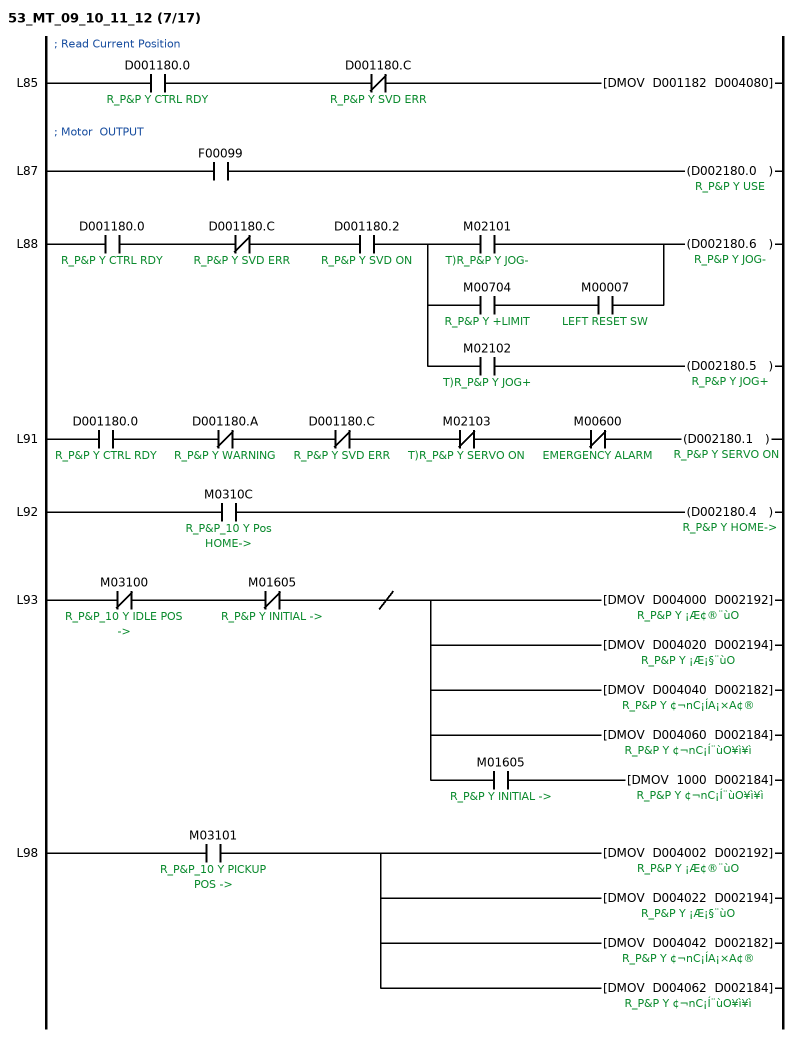
[picture p288: 53_MT_09_10_11_12 rungs L85-L98]
; L85
LOAD      D001180.0	// R_P&P Y CTRL RDY
AND NOT   D001180.C	// R_P&P Y SVD ERR
DMOV      D001182 D004080
// output comment: Read Current Position
//  Motor  OUTPUT
; L87
LOAD      F00099
OUT       D002180.0	// R_P&P Y USE
; L88
LOAD      D001180.0	// R_P&P Y CTRL RDY
AND NOT   D001180.C	// R_P&P Y SVD ERR
AND       D001180.2	// R_P&P Y SVD ON
MPUSH
LOAD      M02101	// T)R_P&P Y JOG-
LOAD      M00704	// R_P&P Y +LIMIT
AND       M00007	// LEFT RESET SW
OR LOAD
AND LOAD
OUT       D002180.6	// R_P&P Y JOG-
MPOP
AND       M02102	// T)R_P&P Y JOG+
OUT       D002180.5	// R_P&P Y JOG+
; L91
LOAD      D001180.0	// R_P&P Y CTRL RDY
AND NOT   D001180.A	// R_P&P Y WARNING
AND NOT   D001180.C	// R_P&P Y SVD ERR
AND NOT   M02103	// T)R_P&P Y SERVO ON
AND NOT   M00600	// EMERGENCY ALARM
OUT       D002180.1	// R_P&P Y SERVO ON
; L92
LOAD      M0310C	// R_P&P_10 Y Pos HOME->
OUT       D002180.4	// R_P&P Y HOME->
; L93
LOAD NOT  M03100	// R_P&P_10 Y IDLE POS ->
AND NOT   M01605	// R_P&P Y INITIAL ->
NOT
DMOV      D004000 D002192	// R_P&P Y ¡Æ¢®¨ùO
DMOV      D004020 D002194	// R_P&P Y ¡Æ¡§¨ùO
DMOV      D004040 D002182	// R_P&P Y ¢¬nC¡ÍA¡×A¢®
DMOV      D004060 D002184	// R_P&P Y ¢¬nC¡Í¨ùO¥ì¥ì
AND       M01605	// R_P&P Y INITIAL ->
DMOV      1000 D002184	// R_P&P Y ¢¬nC¡Í¨ùO¥ì¥ì
; L98
LOAD      M03101	// R_P&P_10 Y PICKUP POS ->
DMOV      D004002 D002192	// R_P&P Y ¡Æ¢®¨ùO
DMOV      D004022 D002194	// R_P&P Y ¡Æ¡§¨ùO
DMOV      D004042 D002182	// R_P&P Y ¢¬nC¡ÍA¡×A¢®
DMOV      D004062 D002184	// R_P&P Y ¢¬nC¡Í¨ùO¥ì¥ì

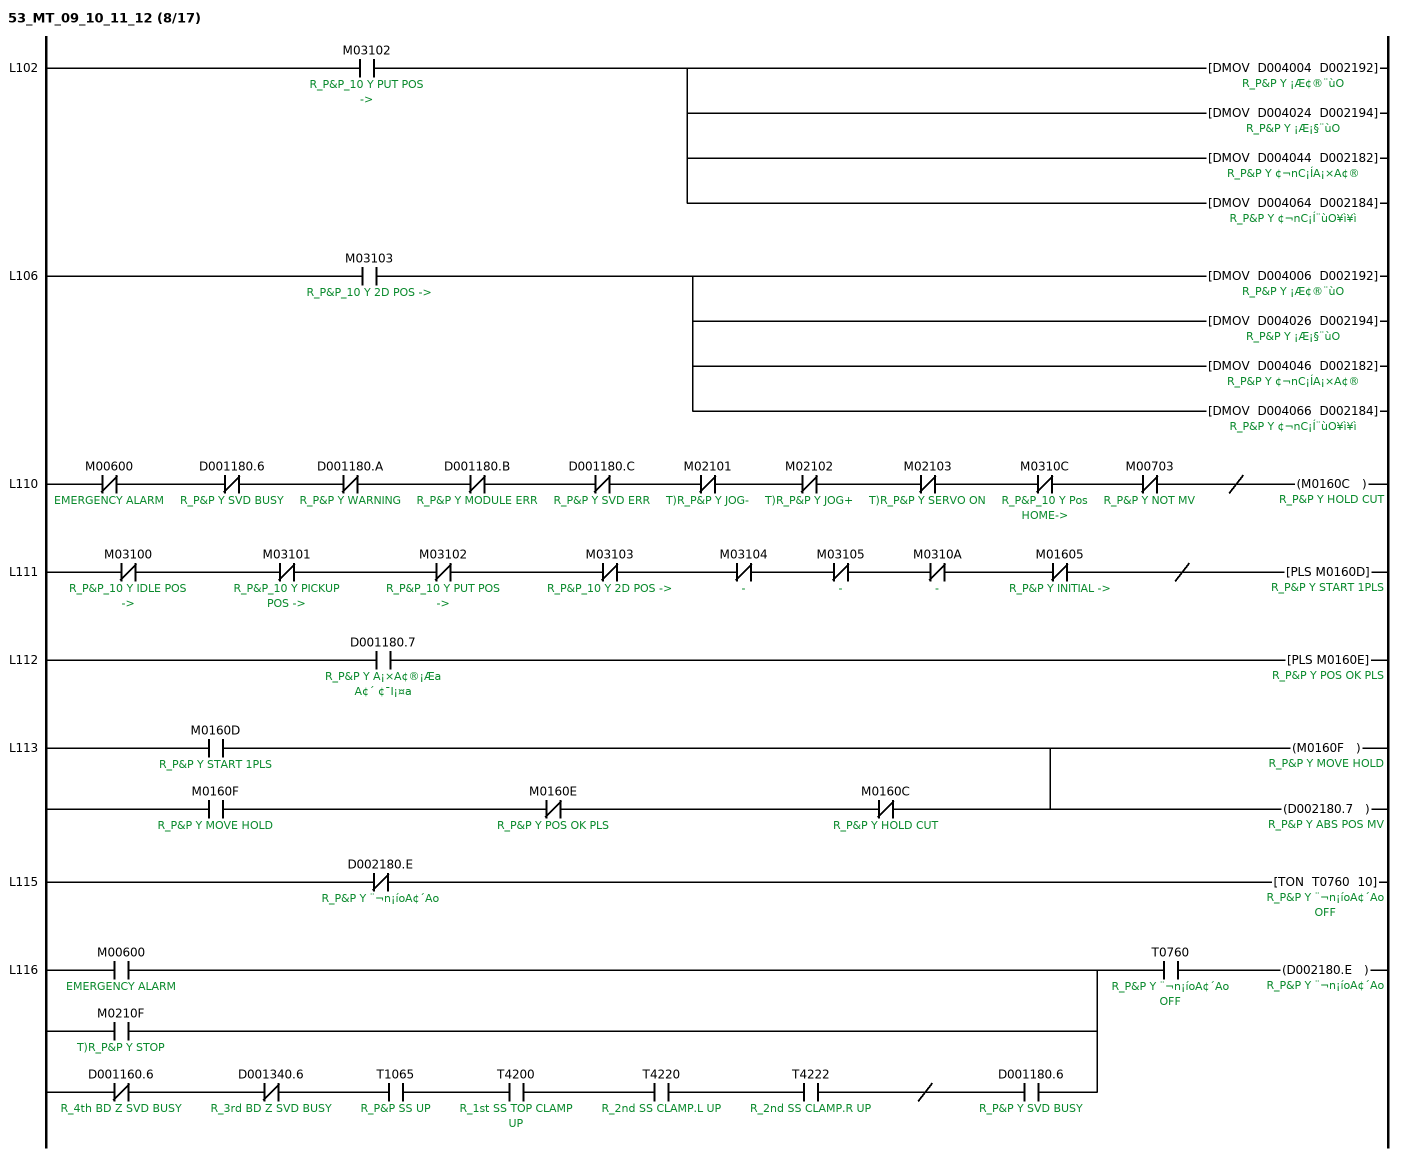
; L102
LOAD      M03102	// R_P&P_10 Y PUT POS ->
DMOV      D004004 D002192	// R_P&P Y ¡Æ¢®¨ùO
DMOV      D004024 D002194	// R_P&P Y ¡Æ¡§¨ùO
DMOV      D004044 D002182	// R_P&P Y ¢¬nC¡ÍA¡×A¢®
DMOV      D004064 D002184	// R_P&P Y ¢¬nC¡Í¨ùO¥ì¥ì
; L106
LOAD      M03103	// R_P&P_10 Y 2D POS ->
DMOV      D004006 D002192	// R_P&P Y ¡Æ¢®¨ùO
DMOV      D004026 D002194	// R_P&P Y ¡Æ¡§¨ùO
DMOV      D004046 D002182	// R_P&P Y ¢¬nC¡ÍA¡×A¢®
DMOV      D004066 D002184	// R_P&P Y ¢¬nC¡Í¨ùO¥ì¥ì
; L110
LOAD NOT  M00600	// EMERGENCY ALARM
AND NOT   D001180.6	// R_P&P Y SVD BUSY
AND NOT   D001180.A	// R_P&P Y WARNING
AND NOT   D001180.B	// R_P&P Y MODULE ERR
AND NOT   D001180.C	// R_P&P Y SVD ERR
AND NOT   M02101	// T)R_P&P Y JOG-
AND NOT   M02102	// T)R_P&P Y JOG+
AND NOT   M02103	// T)R_P&P Y SERVO ON
AND NOT   M0310C	// R_P&P_10 Y Pos HOME->
AND NOT   M00703	// R_P&P Y NOT MV
NOT
OUT       M0160C	// R_P&P Y HOLD CUT
; L111
LOAD NOT  M03100	// R_P&P_10 Y IDLE POS ->
AND NOT   M03101	// R_P&P_10 Y PICKUP POS ->
AND NOT   M03102	// R_P&P_10 Y PUT POS ->
AND NOT   M03103	// R_P&P_10 Y 2D POS ->
AND NOT   M03104	// -
AND NOT   M03105	// -
AND NOT   M0310A	// -
AND NOT   M01605	// R_P&P Y INITIAL ->
NOT
OUTP      M0160D	// R_P&P Y START 1PLS
; L112
LOAD      D001180.7	// R_P&P Y A¡×A¢®¡ÆaA¢´ ¢¯I¡¤a
OUTP      M0160E	// R_P&P Y POS OK PLS
; L113
LOAD      M0160D	// R_P&P Y START 1PLS
LOAD      M0160F	// R_P&P Y MOVE HOLD
AND NOT   M0160E	// R_P&P Y POS OK PLS
AND NOT   M0160C	// R_P&P Y HOLD CUT
OR LOAD
OUT       M0160F	// R_P&P Y MOVE HOLD
OUT       D002180.7	// R_P&P Y ABS POS MV
; L115
LOAD NOT  D002180.E	// R_P&P Y ¨¬n¡íoA¢´Ao
TON       T0760 10	// R_P&P Y ¨¬n¡íoA¢´AoOFF
; L116
LOAD      M00600	// EMERGENCY ALARM
OR        M0210F	// T)R_P&P Y STOP
LOAD NOT  D001160.6	// R_4th BD Z SVD BUSY
AND NOT   D001340.6	// R_3rd BD Z SVD BUSY
AND       T1065	// R_P&P SS UP
AND       T4200	// R_1st SS TOP CLAMP UP
AND       T4220	// R_2nd SS CLAMP.L UP
AND       T4222	// R_2nd SS CLAMP.R UP
NOT
AND       D001180.6	// R_P&P Y SVD BUSY
OR LOAD
AND       T0760	// R_P&P Y ¨¬n¡íoA¢´AoOFF
OUT       D002180.E	// R_P&P Y ¨¬n¡íoA¢´Ao

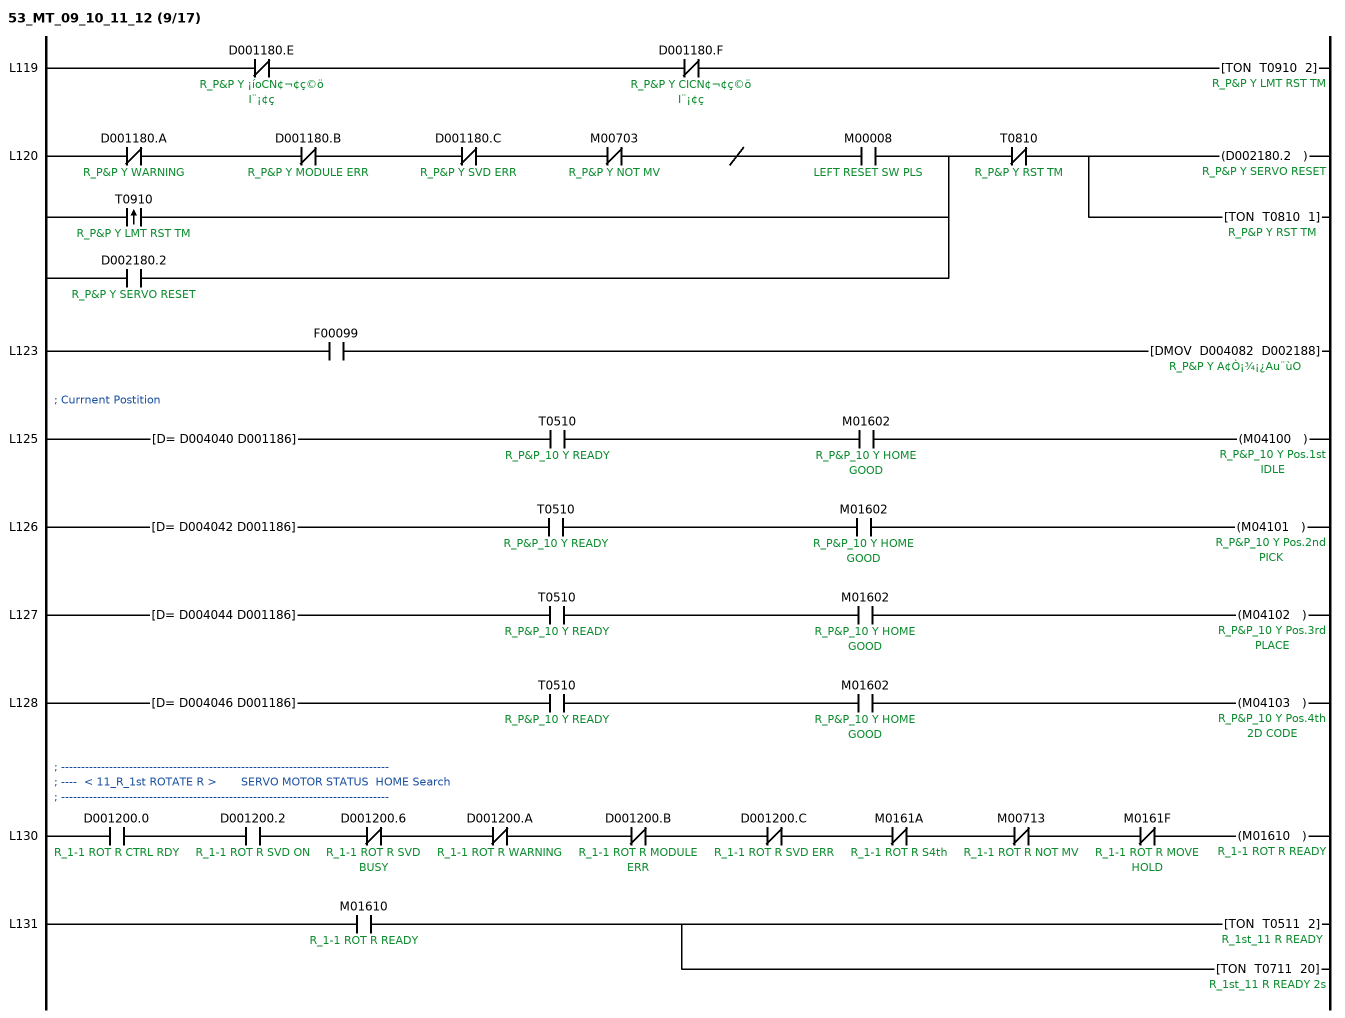
; L119
LOAD NOT  D001180.E	// R_P&P Y ¡íoCN¢¬¢ç©öI¨¡¢ç
AND NOT   D001180.F	// R_P&P Y CICN¢¬¢ç©öI¨¡¢ç
TON       T0910 2	// R_P&P Y LMT RST TM
; L120
LOAD NOT  D001180.A	// R_P&P Y WARNING
AND NOT   D001180.B	// R_P&P Y MODULE ERR
AND NOT   D001180.C	// R_P&P Y SVD ERR
AND NOT   M00703	// R_P&P Y NOT MV
NOT
AND       M00008	// LEFT RESET SW PLS
ORP       T0910	// R_P&P Y LMT RST TM
OR        D002180.2	// R_P&P Y SERVO RESET
AND NOT   T0810	// R_P&P Y RST TM
OUT       D002180.2	// R_P&P Y SERVO RESET
TON       T0810 1	// R_P&P Y RST TM
; L123
LOAD      F00099
DMOV      D004082 D002188	// R_P&P Y A¢Ò¡¾¡¿Au¨ùO
// Currnent Postition
; L125
LOADD=    D004040 D001186
AND       T0510	// R_P&P_10 Y READY
AND       M01602	// R_P&P_10 Y HOME GOOD
OUT       M04100	// R_P&P_10 Y Pos.1st IDLE
; L126
LOADD=    D004042 D001186
AND       T0510	// R_P&P_10 Y READY
AND       M01602	// R_P&P_10 Y HOME GOOD
OUT       M04101	// R_P&P_10 Y Pos.2nd PICK
; L127
LOADD=    D004044 D001186
AND       T0510	// R_P&P_10 Y READY
AND       M01602	// R_P&P_10 Y HOME GOOD
OUT       M04102	// R_P&P_10 Y Pos.3rd PLACE
; L128
LOADD=    D004046 D001186
AND       T0510	// R_P&P_10 Y READY
AND       M01602	// R_P&P_10 Y HOME GOOD
OUT       M04103	// R_P&P_10 Y Pos.4th 2D CODE
// ----------------------------------------------------------------------------------
// 
// ----  < 11_R_1st ROTATE R >       SERVO MOTOR STATUS  HOME Search
// 
// ----------------------------------------------------------------------------------
; L130
LOAD      D001200.0	// R_1-1 ROT R CTRL RDY
AND       D001200.2	// R_1-1 ROT R SVD ON
AND NOT   D001200.6	// R_1-1 ROT R SVD BUSY
AND NOT   D001200.A	// R_1-1 ROT R WARNING
AND NOT   D001200.B	// R_1-1 ROT R MODULE ERR
AND NOT   D001200.C	// R_1-1 ROT R SVD ERR
AND NOT   M0161A	// R_1-1 ROT R S4th
AND NOT   M00713	// R_1-1 ROT R NOT MV
AND NOT   M0161F	// R_1-1 ROT R MOVE HOLD
OUT       M01610	// R_1-1 ROT R READY
; L131
LOAD      M01610	// R_1-1 ROT R READY
TON       T0511 2	// R_1st_11 R READY
TON       T0711 20	// R_1st_11 R READY 2s

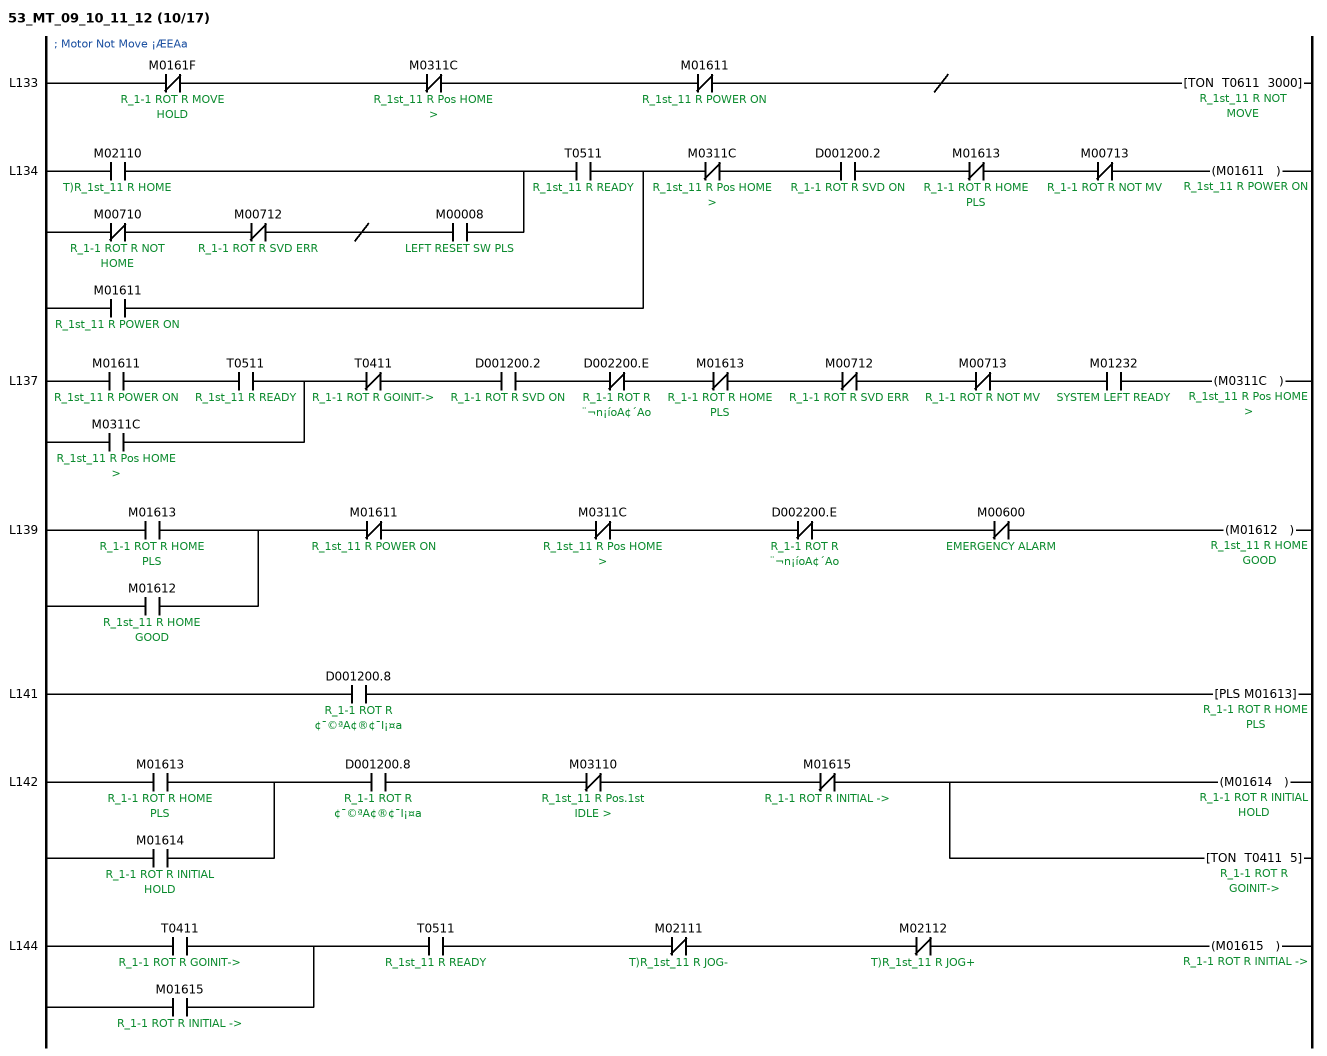
; L133
LOAD NOT  M0161F	// R_1-1 ROT R MOVE HOLD
AND NOT   M0311C	// R_1st_11 R Pos HOME >
AND NOT   M01611	// R_1st_11 R POWER ON
NOT
TON       T0611 3000	// R_1st_11 R NOT MOVE
// output comment: Motor Not Move ¡ÆEAa
; L134
LOAD      M02110	// T)R_1st_11 R HOME
LOAD NOT  M00710	// R_1-1 ROT R NOT HOME
AND NOT   M00712	// R_1-1 ROT R SVD ERR
NOT
AND       M00008	// LEFT RESET SW PLS
OR LOAD
AND       T0511	// R_1st_11 R READY
OR        M01611	// R_1st_11 R POWER ON
AND NOT   M0311C	// R_1st_11 R Pos HOME >
AND       D001200.2	// R_1-1 ROT R SVD ON
AND NOT   M01613	// R_1-1 ROT R HOME PLS
AND NOT   M00713	// R_1-1 ROT R NOT MV
OUT       M01611	// R_1st_11 R POWER ON
; L137
LOAD      M01611	// R_1st_11 R POWER ON
AND       T0511	// R_1st_11 R READY
OR        M0311C	// R_1st_11 R Pos HOME >
AND NOT   T0411	// R_1-1 ROT R GOINIT->
AND       D001200.2	// R_1-1 ROT R SVD ON
AND NOT   D002200.E	// R_1-1 ROT R ¨¬n¡íoA¢´Ao
AND NOT   M01613	// R_1-1 ROT R HOME PLS
AND NOT   M00712	// R_1-1 ROT R SVD ERR
AND NOT   M00713	// R_1-1 ROT R NOT MV
AND       M01232	// SYSTEM LEFT READY
OUT       M0311C	// R_1st_11 R Pos HOME >
; L139
LOAD      M01613	// R_1-1 ROT R HOME PLS
OR        M01612	// R_1st_11 R HOME GOOD
AND NOT   M01611	// R_1st_11 R POWER ON
AND NOT   M0311C	// R_1st_11 R Pos HOME >
AND NOT   D002200.E	// R_1-1 ROT R ¨¬n¡íoA¢´Ao
AND NOT   M00600	// EMERGENCY ALARM
OUT       M01612	// R_1st_11 R HOME GOOD
; L141
LOAD      D001200.8	// R_1-1 ROT R ¢¯©ªA¢®¢¯I¡¤a
OUTP      M01613	// R_1-1 ROT R HOME PLS
; L142
LOAD      M01613	// R_1-1 ROT R HOME PLS
OR        M01614	// R_1-1 ROT R INITIAL HOLD
AND       D001200.8	// R_1-1 ROT R ¢¯©ªA¢®¢¯I¡¤a
AND NOT   M03110	// R_1st_11 R Pos.1st IDLE >
AND NOT   M01615	// R_1-1 ROT R INITIAL ->
OUT       M01614	// R_1-1 ROT R INITIAL HOLD
TON       T0411 5	// R_1-1 ROT R GOINIT->
; L144
LOAD      T0411	// R_1-1 ROT R GOINIT->
OR        M01615	// R_1-1 ROT R INITIAL ->
AND       T0511	// R_1st_11 R READY
AND NOT   M02111	// T)R_1st_11 R JOG-
AND NOT   M02112	// T)R_1st_11 R JOG+
OUT       M01615	// R_1-1 ROT R INITIAL ->

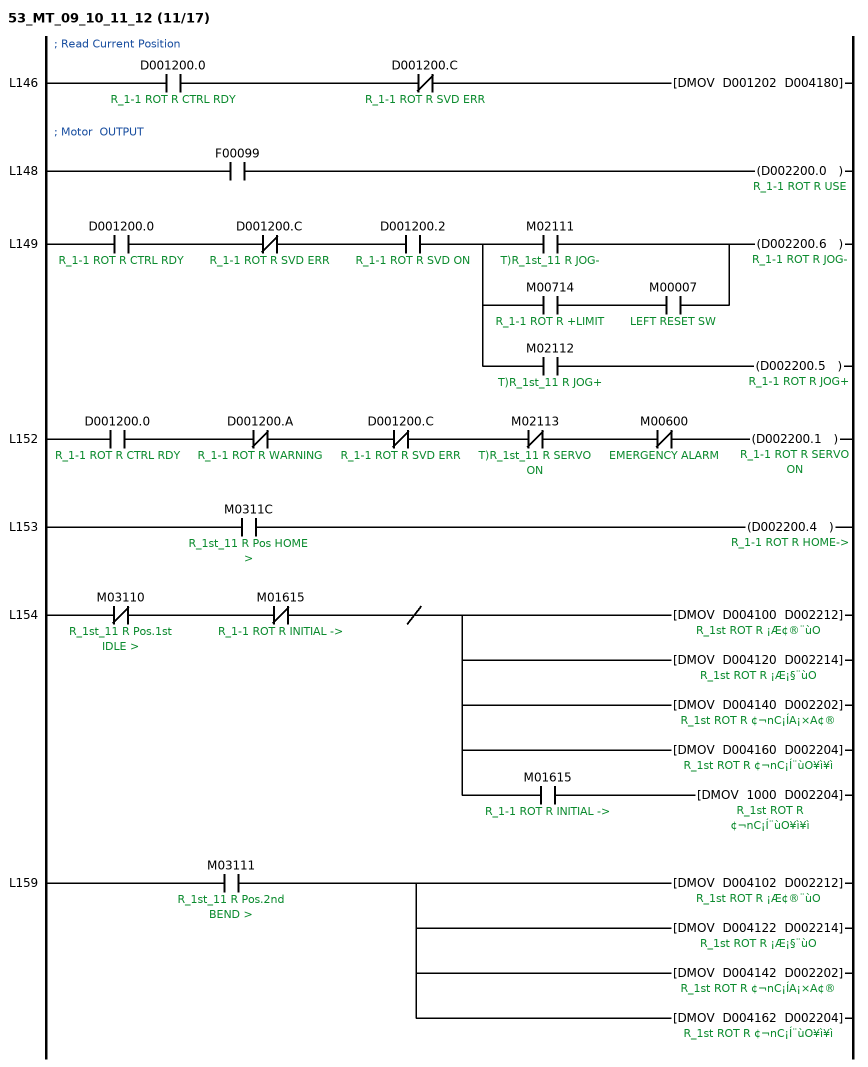
; L146
LOAD      D001200.0	// R_1-1 ROT R CTRL RDY
AND NOT   D001200.C	// R_1-1 ROT R SVD ERR
DMOV      D001202 D004180
// output comment: Read Current Position
//  Motor  OUTPUT
; L148
LOAD      F00099
OUT       D002200.0	// R_1-1 ROT R USE
; L149
LOAD      D001200.0	// R_1-1 ROT R CTRL RDY
AND NOT   D001200.C	// R_1-1 ROT R SVD ERR
AND       D001200.2	// R_1-1 ROT R SVD ON
MPUSH
LOAD      M02111	// T)R_1st_11 R JOG-
LOAD      M00714	// R_1-1 ROT R +LIMIT
AND       M00007	// LEFT RESET SW
OR LOAD
AND LOAD
OUT       D002200.6	// R_1-1 ROT R JOG-
MPOP
AND       M02112	// T)R_1st_11 R JOG+
OUT       D002200.5	// R_1-1 ROT R JOG+
; L152
LOAD      D001200.0	// R_1-1 ROT R CTRL RDY
AND NOT   D001200.A	// R_1-1 ROT R WARNING
AND NOT   D001200.C	// R_1-1 ROT R SVD ERR
AND NOT   M02113	// T)R_1st_11 R SERVO ON
AND NOT   M00600	// EMERGENCY ALARM
OUT       D002200.1	// R_1-1 ROT R SERVO ON
; L153
LOAD      M0311C	// R_1st_11 R Pos HOME >
OUT       D002200.4	// R_1-1 ROT R HOME->
; L154
LOAD NOT  M03110	// R_1st_11 R Pos.1st IDLE >
AND NOT   M01615	// R_1-1 ROT R INITIAL ->
NOT
DMOV      D004100 D002212	// R_1st ROT R ¡Æ¢®¨ùO
DMOV      D004120 D002214	// R_1st ROT R ¡Æ¡§¨ùO
DMOV      D004140 D002202	// R_1st ROT R ¢¬nC¡ÍA¡×A¢®
DMOV      D004160 D002204	// R_1st ROT R ¢¬nC¡Í¨ùO¥ì¥ì
AND       M01615	// R_1-1 ROT R INITIAL ->
DMOV      1000 D002204	// R_1st ROT R ¢¬nC¡Í¨ùO¥ì¥ì
; L159
LOAD      M03111	// R_1st_11 R Pos.2nd BEND >
DMOV      D004102 D002212	// R_1st ROT R ¡Æ¢®¨ùO
DMOV      D004122 D002214	// R_1st ROT R ¡Æ¡§¨ùO
DMOV      D004142 D002202	// R_1st ROT R ¢¬nC¡ÍA¡×A¢®
DMOV      D004162 D002204	// R_1st ROT R ¢¬nC¡Í¨ùO¥ì¥ì

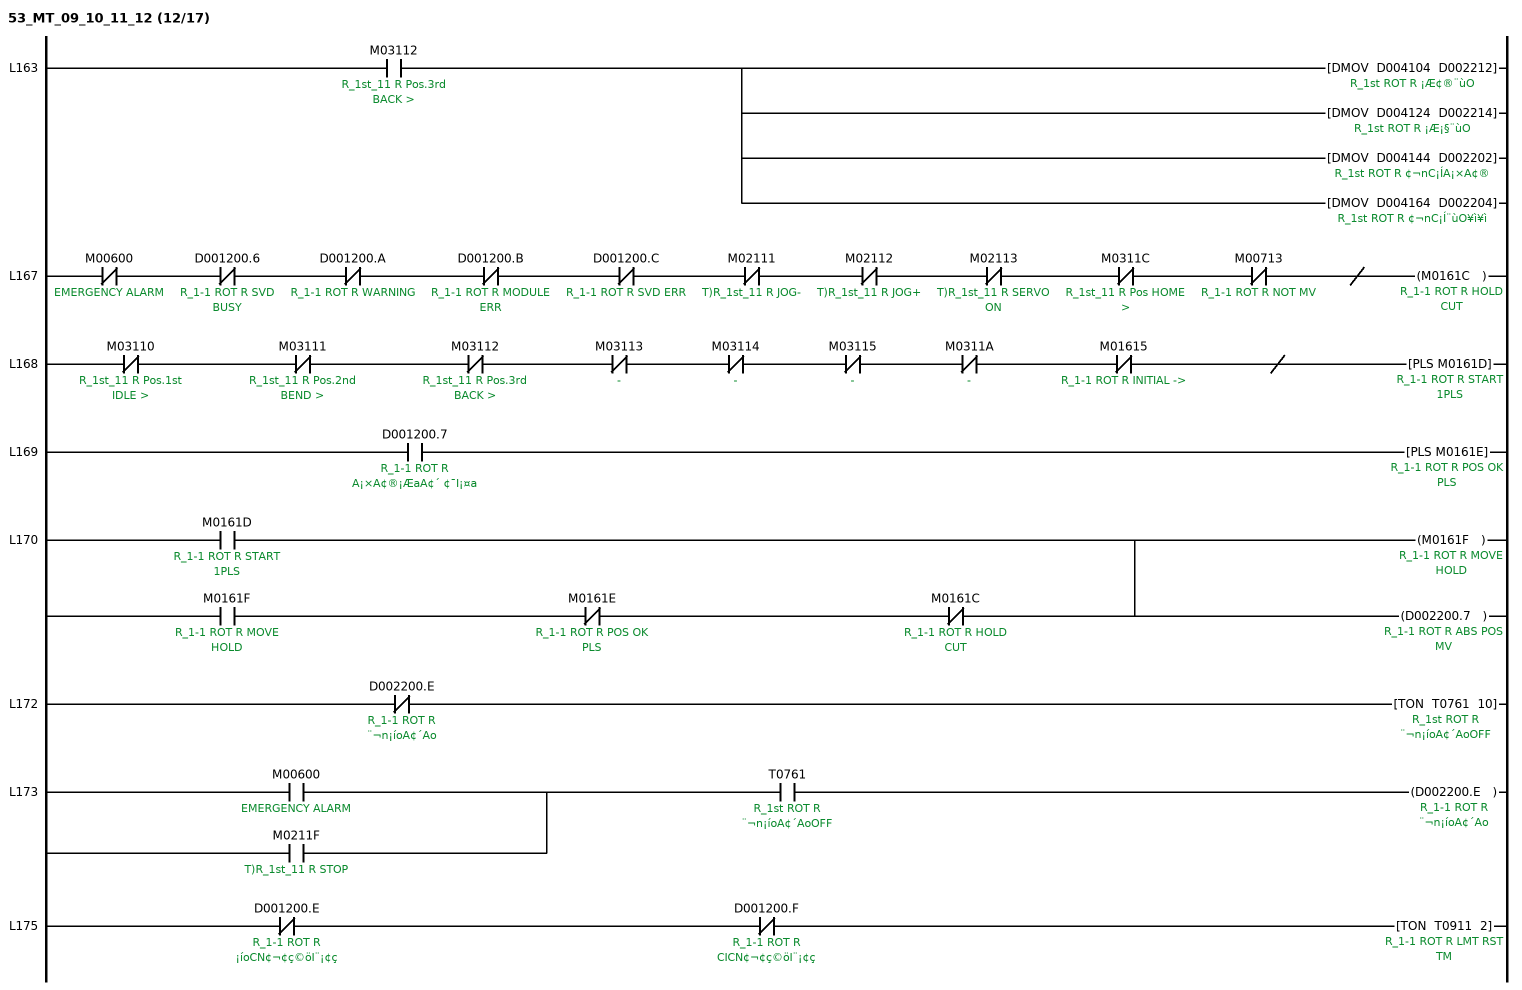
; L163
LOAD      M03112	// R_1st_11 R Pos.3rd BACK >
DMOV      D004104 D002212	// R_1st ROT R ¡Æ¢®¨ùO
DMOV      D004124 D002214	// R_1st ROT R ¡Æ¡§¨ùO
DMOV      D004144 D002202	// R_1st ROT R ¢¬nC¡ÍA¡×A¢®
DMOV      D004164 D002204	// R_1st ROT R ¢¬nC¡Í¨ùO¥ì¥ì
; L167
LOAD NOT  M00600	// EMERGENCY ALARM
AND NOT   D001200.6	// R_1-1 ROT R SVD BUSY
AND NOT   D001200.A	// R_1-1 ROT R WARNING
AND NOT   D001200.B	// R_1-1 ROT R MODULE ERR
AND NOT   D001200.C	// R_1-1 ROT R SVD ERR
AND NOT   M02111	// T)R_1st_11 R JOG-
AND NOT   M02112	// T)R_1st_11 R JOG+
AND NOT   M02113	// T)R_1st_11 R SERVO ON
AND NOT   M0311C	// R_1st_11 R Pos HOME >
AND NOT   M00713	// R_1-1 ROT R NOT MV
NOT
OUT       M0161C	// R_1-1 ROT R HOLD CUT
; L168
LOAD NOT  M03110	// R_1st_11 R Pos.1st IDLE >
AND NOT   M03111	// R_1st_11 R Pos.2nd BEND >
AND NOT   M03112	// R_1st_11 R Pos.3rd BACK >
AND NOT   M03113	// -
AND NOT   M03114	// -
AND NOT   M03115	// -
AND NOT   M0311A	// -
AND NOT   M01615	// R_1-1 ROT R INITIAL ->
NOT
OUTP      M0161D	// R_1-1 ROT R START 1PLS
; L169
LOAD      D001200.7	// R_1-1 ROT R A¡×A¢®¡ÆaA¢´ ¢¯I¡¤a
OUTP      M0161E	// R_1-1 ROT R POS OK PLS
; L170
LOAD      M0161D	// R_1-1 ROT R START 1PLS
LOAD      M0161F	// R_1-1 ROT R MOVE HOLD
AND NOT   M0161E	// R_1-1 ROT R POS OK PLS
AND NOT   M0161C	// R_1-1 ROT R HOLD CUT
OR LOAD
OUT       M0161F	// R_1-1 ROT R MOVE HOLD
OUT       D002200.7	// R_1-1 ROT R ABS POS MV
; L172
LOAD NOT  D002200.E	// R_1-1 ROT R ¨¬n¡íoA¢´Ao
TON       T0761 10	// R_1st ROT R ¨¬n¡íoA¢´AoOFF
; L173
LOAD      M00600	// EMERGENCY ALARM
OR        M0211F	// T)R_1st_11 R STOP
AND       T0761	// R_1st ROT R ¨¬n¡íoA¢´AoOFF
OUT       D002200.E	// R_1-1 ROT R ¨¬n¡íoA¢´Ao
; L175
LOAD NOT  D001200.E	// R_1-1 ROT R ¡íoCN¢¬¢ç©öI¨¡¢ç
AND NOT   D001200.F	// R_1-1 ROT R CICN¢¬¢ç©öI¨¡¢ç
TON       T0911 2	// R_1-1 ROT R LMT RST TM

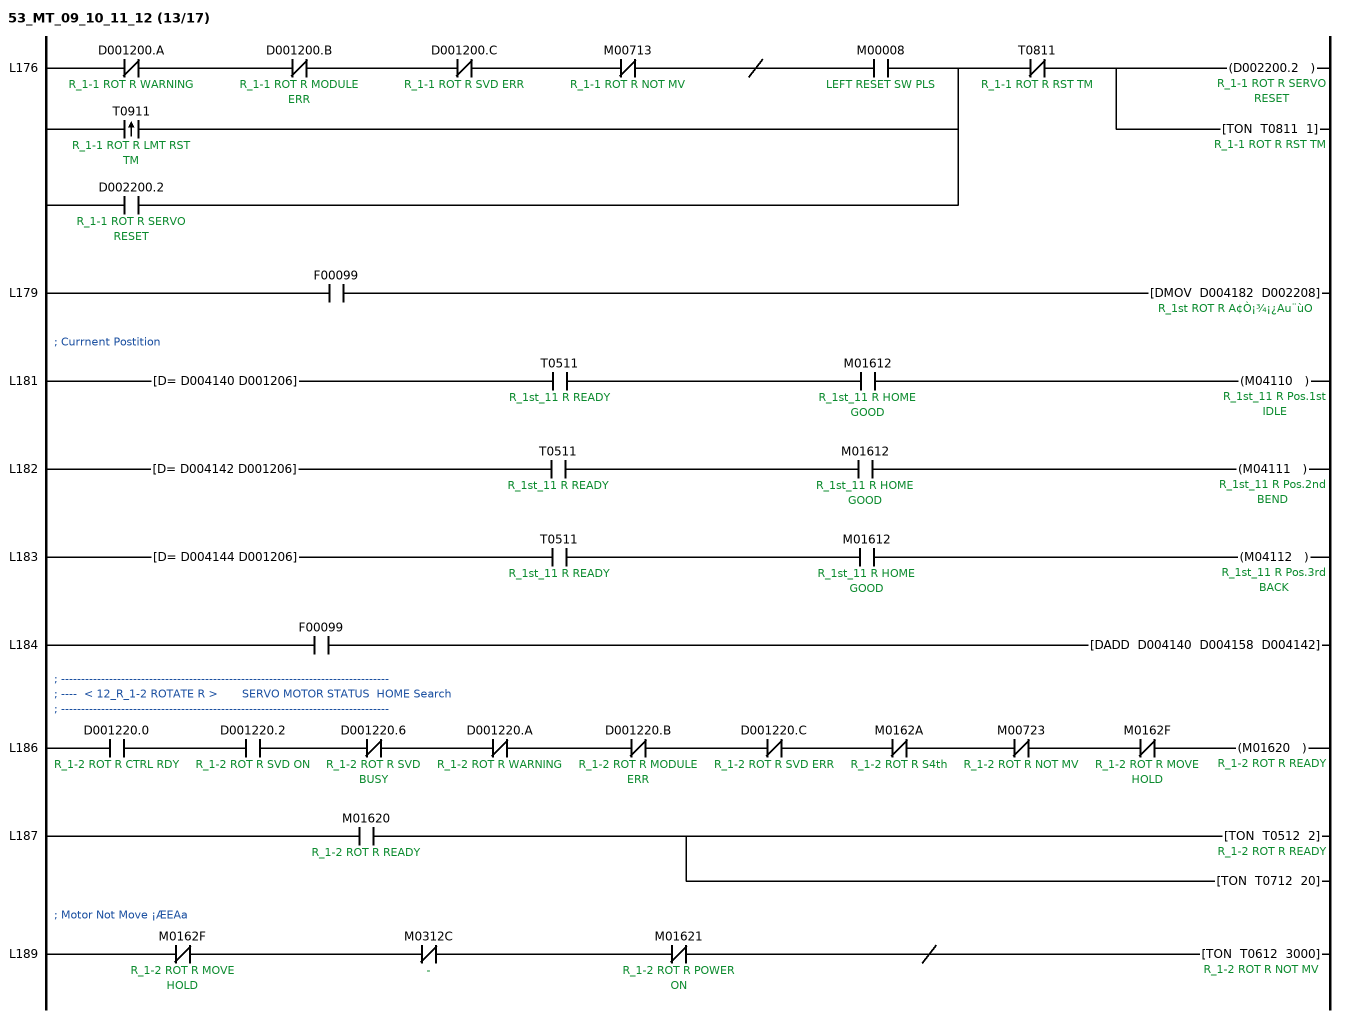
; L176
LOAD NOT  D001200.A	// R_1-1 ROT R WARNING
AND NOT   D001200.B	// R_1-1 ROT R MODULE ERR
AND NOT   D001200.C	// R_1-1 ROT R SVD ERR
AND NOT   M00713	// R_1-1 ROT R NOT MV
NOT
AND       M00008	// LEFT RESET SW PLS
ORP       T0911	// R_1-1 ROT R LMT RST TM
OR        D002200.2	// R_1-1 ROT R SERVO RESET
AND NOT   T0811	// R_1-1 ROT R RST TM
OUT       D002200.2	// R_1-1 ROT R SERVO RESET
TON       T0811 1	// R_1-1 ROT R RST TM
; L179
LOAD      F00099
DMOV      D004182 D002208	// R_1st ROT R A¢Ò¡¾¡¿Au¨ùO
// Currnent Postition
; L181
LOADD=    D004140 D001206
AND       T0511	// R_1st_11 R READY
AND       M01612	// R_1st_11 R HOME GOOD
OUT       M04110	// R_1st_11 R Pos.1st IDLE
; L182
LOADD=    D004142 D001206
AND       T0511	// R_1st_11 R READY
AND       M01612	// R_1st_11 R HOME GOOD
OUT       M04111	// R_1st_11 R Pos.2nd BEND
; L183
LOADD=    D004144 D001206
AND       T0511	// R_1st_11 R READY
AND       M01612	// R_1st_11 R HOME GOOD
OUT       M04112	// R_1st_11 R Pos.3rd BACK
; L184
LOAD      F00099
DADD      D004140 D004158 D004142
// ----------------------------------------------------------------------------------
// 
// ----  < 12_R_1-2 ROTATE R >       SERVO MOTOR STATUS  HOME Search
// 
// ----------------------------------------------------------------------------------
; L186
LOAD      D001220.0	// R_1-2 ROT R CTRL RDY
AND       D001220.2	// R_1-2 ROT R SVD ON
AND NOT   D001220.6	// R_1-2 ROT R SVD BUSY
AND NOT   D001220.A	// R_1-2 ROT R WARNING
AND NOT   D001220.B	// R_1-2 ROT R MODULE ERR
AND NOT   D001220.C	// R_1-2 ROT R SVD ERR
AND NOT   M0162A	// R_1-2 ROT R S4th
AND NOT   M00723	// R_1-2 ROT R NOT MV
AND NOT   M0162F	// R_1-2 ROT R MOVE HOLD
OUT       M01620	// R_1-2 ROT R READY
; L187
LOAD      M01620	// R_1-2 ROT R READY
TON       T0512 2	// R_1-2 ROT R READY
TON       T0712 20
; L189
LOAD NOT  M0162F	// R_1-2 ROT R MOVE HOLD
AND NOT   M0312C	// -
AND NOT   M01621	// R_1-2 ROT R POWER ON
NOT
TON       T0612 3000	// R_1-2 ROT R NOT MV
// output comment: Motor Not Move ¡ÆEAa

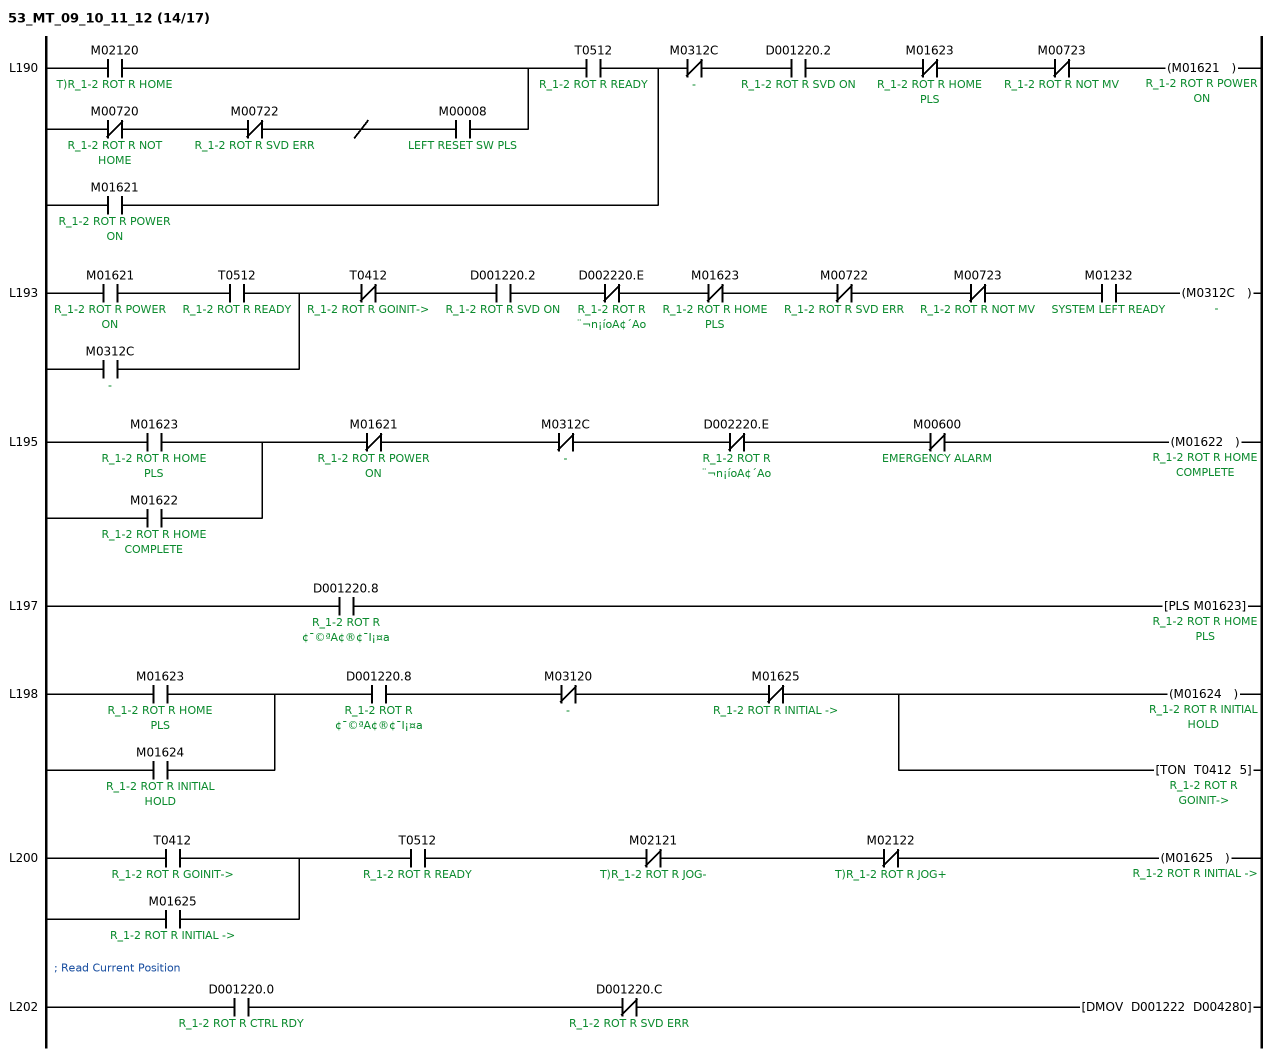
; L190
LOAD      M02120	// T)R_1-2 ROT R HOME
LOAD NOT  M00720	// R_1-2 ROT R NOT HOME
AND NOT   M00722	// R_1-2 ROT R SVD ERR
NOT
AND       M00008	// LEFT RESET SW PLS
OR LOAD
AND       T0512	// R_1-2 ROT R READY
OR        M01621	// R_1-2 ROT R POWER ON
AND NOT   M0312C	// -
AND       D001220.2	// R_1-2 ROT R SVD ON
AND NOT   M01623	// R_1-2 ROT R HOME PLS
AND NOT   M00723	// R_1-2 ROT R NOT MV
OUT       M01621	// R_1-2 ROT R POWER ON
; L193
LOAD      M01621	// R_1-2 ROT R POWER ON
AND       T0512	// R_1-2 ROT R READY
OR        M0312C	// -
AND NOT   T0412	// R_1-2 ROT R GOINIT->
AND       D001220.2	// R_1-2 ROT R SVD ON
AND NOT   D002220.E	// R_1-2 ROT R ¨¬n¡íoA¢´Ao
AND NOT   M01623	// R_1-2 ROT R HOME PLS
AND NOT   M00722	// R_1-2 ROT R SVD ERR
AND NOT   M00723	// R_1-2 ROT R NOT MV
AND       M01232	// SYSTEM LEFT READY
OUT       M0312C	// -
; L195
LOAD      M01623	// R_1-2 ROT R HOME PLS
OR        M01622	// R_1-2 ROT R HOME COMPLETE
AND NOT   M01621	// R_1-2 ROT R POWER ON
AND NOT   M0312C	// -
AND NOT   D002220.E	// R_1-2 ROT R ¨¬n¡íoA¢´Ao
AND NOT   M00600	// EMERGENCY ALARM
OUT       M01622	// R_1-2 ROT R HOME COMPLETE
; L197
LOAD      D001220.8	// R_1-2 ROT R ¢¯©ªA¢®¢¯I¡¤a
OUTP      M01623	// R_1-2 ROT R HOME PLS
; L198
LOAD      M01623	// R_1-2 ROT R HOME PLS
OR        M01624	// R_1-2 ROT R INITIAL HOLD
AND       D001220.8	// R_1-2 ROT R ¢¯©ªA¢®¢¯I¡¤a
AND NOT   M03120	// -
AND NOT   M01625	// R_1-2 ROT R INITIAL ->
OUT       M01624	// R_1-2 ROT R INITIAL HOLD
TON       T0412 5	// R_1-2 ROT R GOINIT->
; L200
LOAD      T0412	// R_1-2 ROT R GOINIT->
OR        M01625	// R_1-2 ROT R INITIAL ->
AND       T0512	// R_1-2 ROT R READY
AND NOT   M02121	// T)R_1-2 ROT R JOG-
AND NOT   M02122	// T)R_1-2 ROT R JOG+
OUT       M01625	// R_1-2 ROT R INITIAL ->
; L202
LOAD      D001220.0	// R_1-2 ROT R CTRL RDY
AND NOT   D001220.C	// R_1-2 ROT R SVD ERR
DMOV      D001222 D004280
// output comment: Read Current Position

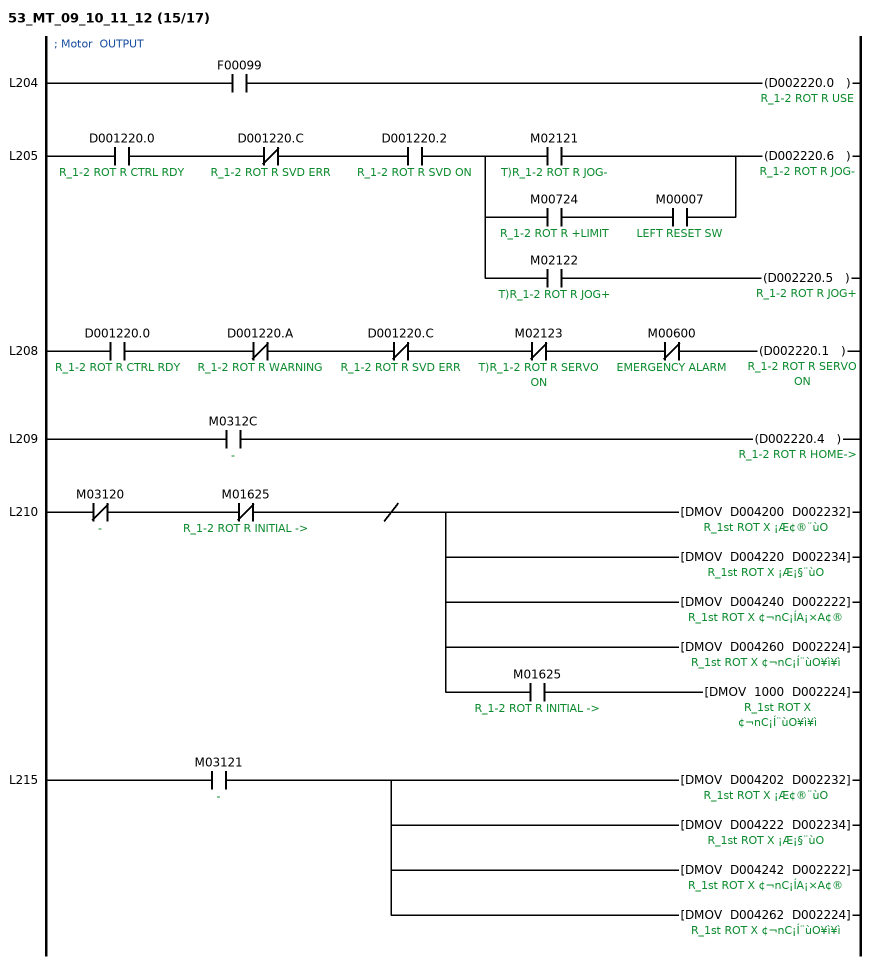
//  Motor  OUTPUT
; L204
LOAD      F00099
OUT       D002220.0	// R_1-2 ROT R USE
; L205
LOAD      D001220.0	// R_1-2 ROT R CTRL RDY
AND NOT   D001220.C	// R_1-2 ROT R SVD ERR
AND       D001220.2	// R_1-2 ROT R SVD ON
MPUSH
LOAD      M02121	// T)R_1-2 ROT R JOG-
LOAD      M00724	// R_1-2 ROT R +LIMIT
AND       M00007	// LEFT RESET SW
OR LOAD
AND LOAD
OUT       D002220.6	// R_1-2 ROT R JOG-
MPOP
AND       M02122	// T)R_1-2 ROT R JOG+
OUT       D002220.5	// R_1-2 ROT R JOG+
; L208
LOAD      D001220.0	// R_1-2 ROT R CTRL RDY
AND NOT   D001220.A	// R_1-2 ROT R WARNING
AND NOT   D001220.C	// R_1-2 ROT R SVD ERR
AND NOT   M02123	// T)R_1-2 ROT R SERVO ON
AND NOT   M00600	// EMERGENCY ALARM
OUT       D002220.1	// R_1-2 ROT R SERVO ON
; L209
LOAD      M0312C	// -
OUT       D002220.4	// R_1-2 ROT R HOME->
; L210
LOAD NOT  M03120	// -
AND NOT   M01625	// R_1-2 ROT R INITIAL ->
NOT
DMOV      D004200 D002232	// R_1st ROT X ¡Æ¢®¨ùO
DMOV      D004220 D002234	// R_1st ROT X ¡Æ¡§¨ùO
DMOV      D004240 D002222	// R_1st ROT X ¢¬nC¡ÍA¡×A¢®
DMOV      D004260 D002224	// R_1st ROT X ¢¬nC¡Í¨ùO¥ì¥ì
AND       M01625	// R_1-2 ROT R INITIAL ->
DMOV      1000 D002224	// R_1st ROT X ¢¬nC¡Í¨ùO¥ì¥ì
; L215
LOAD      M03121	// -
DMOV      D004202 D002232	// R_1st ROT X ¡Æ¢®¨ùO
DMOV      D004222 D002234	// R_1st ROT X ¡Æ¡§¨ùO
DMOV      D004242 D002222	// R_1st ROT X ¢¬nC¡ÍA¡×A¢®
DMOV      D004262 D002224	// R_1st ROT X ¢¬nC¡Í¨ùO¥ì¥ì

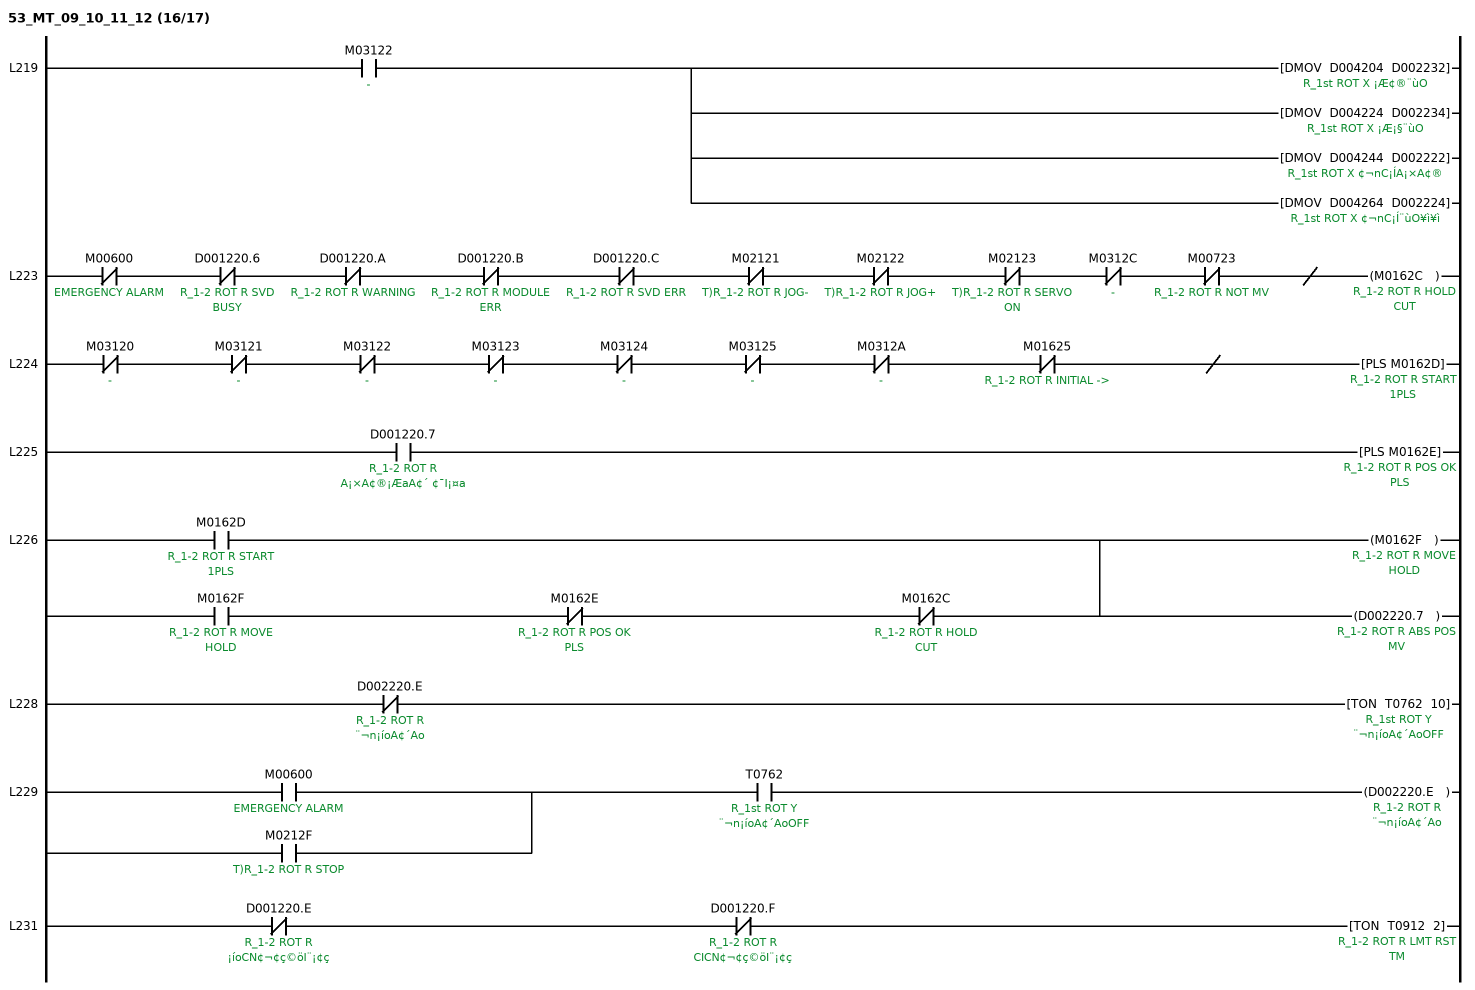
; L219
LOAD      M03122	// -
DMOV      D004204 D002232	// R_1st ROT X ¡Æ¢®¨ùO
DMOV      D004224 D002234	// R_1st ROT X ¡Æ¡§¨ùO
DMOV      D004244 D002222	// R_1st ROT X ¢¬nC¡ÍA¡×A¢®
DMOV      D004264 D002224	// R_1st ROT X ¢¬nC¡Í¨ùO¥ì¥ì
; L223
LOAD NOT  M00600	// EMERGENCY ALARM
AND NOT   D001220.6	// R_1-2 ROT R SVD BUSY
AND NOT   D001220.A	// R_1-2 ROT R WARNING
AND NOT   D001220.B	// R_1-2 ROT R MODULE ERR
AND NOT   D001220.C	// R_1-2 ROT R SVD ERR
AND NOT   M02121	// T)R_1-2 ROT R JOG-
AND NOT   M02122	// T)R_1-2 ROT R JOG+
AND NOT   M02123	// T)R_1-2 ROT R SERVO ON
AND NOT   M0312C	// -
AND NOT   M00723	// R_1-2 ROT R NOT MV
NOT
OUT       M0162C	// R_1-2 ROT R HOLD CUT
; L224
LOAD NOT  M03120	// -
AND NOT   M03121	// -
AND NOT   M03122	// -
AND NOT   M03123	// -
AND NOT   M03124	// -
AND NOT   M03125	// -
AND NOT   M0312A	// -
AND NOT   M01625	// R_1-2 ROT R INITIAL ->
NOT
OUTP      M0162D	// R_1-2 ROT R START 1PLS
; L225
LOAD      D001220.7	// R_1-2 ROT R A¡×A¢®¡ÆaA¢´ ¢¯I¡¤a
OUTP      M0162E	// R_1-2 ROT R POS OK PLS
; L226
LOAD      M0162D	// R_1-2 ROT R START 1PLS
LOAD      M0162F	// R_1-2 ROT R MOVE HOLD
AND NOT   M0162E	// R_1-2 ROT R POS OK PLS
AND NOT   M0162C	// R_1-2 ROT R HOLD CUT
OR LOAD
OUT       M0162F	// R_1-2 ROT R MOVE HOLD
OUT       D002220.7	// R_1-2 ROT R ABS POS MV
; L228
LOAD NOT  D002220.E	// R_1-2 ROT R ¨¬n¡íoA¢´Ao
TON       T0762 10	// R_1st ROT Y ¨¬n¡íoA¢´AoOFF
; L229
LOAD      M00600	// EMERGENCY ALARM
OR        M0212F	// T)R_1-2 ROT R STOP
AND       T0762	// R_1st ROT Y ¨¬n¡íoA¢´AoOFF
OUT       D002220.E	// R_1-2 ROT R ¨¬n¡íoA¢´Ao
; L231
LOAD NOT  D001220.E	// R_1-2 ROT R ¡íoCN¢¬¢ç©öI¨¡¢ç
AND NOT   D001220.F	// R_1-2 ROT R CICN¢¬¢ç©öI¨¡¢ç
TON       T0912 2	// R_1-2 ROT R LMT RST TM

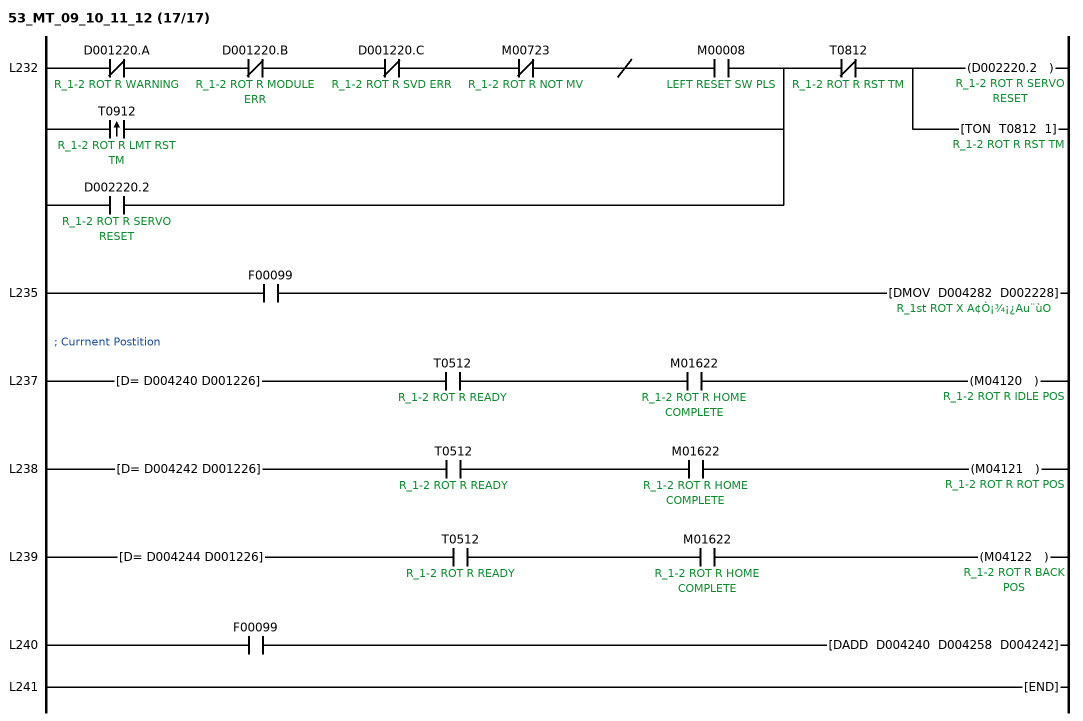
; L232
LOAD NOT  D001220.A	// R_1-2 ROT R WARNING
AND NOT   D001220.B	// R_1-2 ROT R MODULE ERR
AND NOT   D001220.C	// R_1-2 ROT R SVD ERR
AND NOT   M00723	// R_1-2 ROT R NOT MV
NOT
AND       M00008	// LEFT RESET SW PLS
ORP       T0912	// R_1-2 ROT R LMT RST TM
OR        D002220.2	// R_1-2 ROT R SERVO RESET
AND NOT   T0812	// R_1-2 ROT R RST TM
OUT       D002220.2	// R_1-2 ROT R SERVO RESET
TON       T0812 1	// R_1-2 ROT R RST TM
; L235
LOAD      F00099
DMOV      D004282 D002228	// R_1st ROT X A¢Ò¡¾¡¿Au¨ùO
// Currnent Postition
; L237
LOADD=    D004240 D001226
AND       T0512	// R_1-2 ROT R READY
AND       M01622	// R_1-2 ROT R HOME COMPLETE
OUT       M04120	// R_1-2 ROT R IDLE POS
; L238
LOADD=    D004242 D001226
AND       T0512	// R_1-2 ROT R READY
AND       M01622	// R_1-2 ROT R HOME COMPLETE
OUT       M04121	// R_1-2 ROT R ROT POS
; L239
LOADD=    D004244 D001226
AND       T0512	// R_1-2 ROT R READY
AND       M01622	// R_1-2 ROT R HOME COMPLETE
OUT       M04122	// R_1-2 ROT R BACK POS
; L240
LOAD      F00099
DADD      D004240 D004258 D004242
; L241
END

PROGRAM 54_MT_13_14_15_16 (task: ¨ö¨¬A¥ì CA¡¤I¡¾¡¿¡¤¡Í)

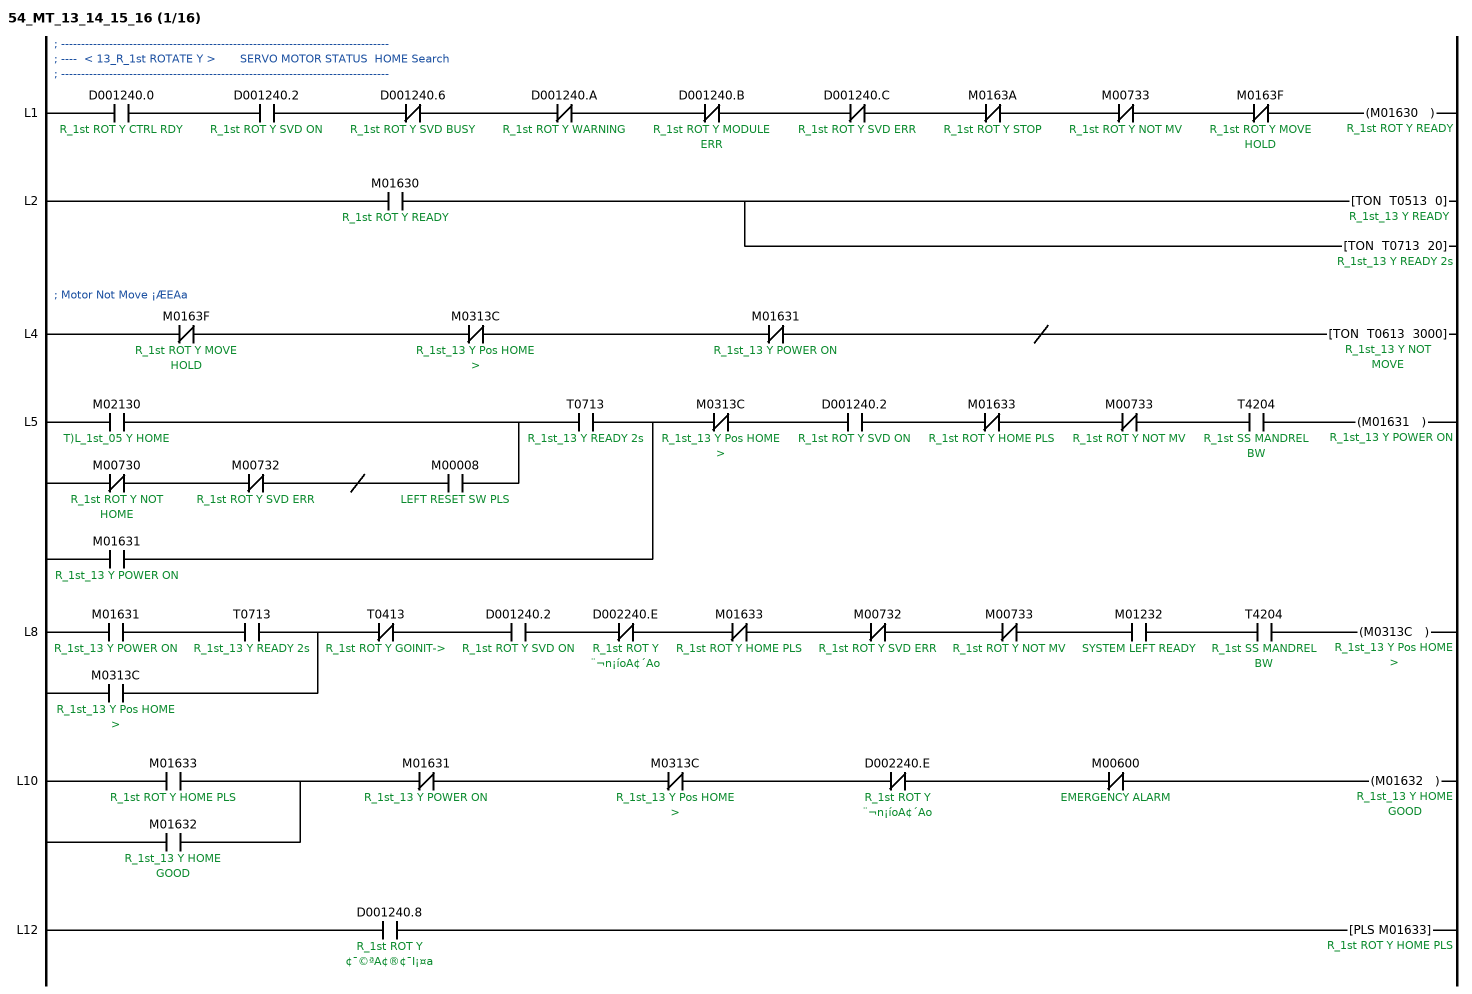
// ----------------------------------------------------------------------------------
// 
// ----  < 13_R_1st ROTATE Y >       SERVO MOTOR STATUS  HOME Search
// 
// ----------------------------------------------------------------------------------
; L1
LOAD      D001240.0	// R_1st ROT Y CTRL RDY
AND       D001240.2	// R_1st ROT Y SVD ON
AND NOT   D001240.6	// R_1st ROT Y SVD BUSY
AND NOT   D001240.A	// R_1st ROT Y WARNING
AND NOT   D001240.B	// R_1st ROT Y MODULE ERR
AND NOT   D001240.C	// R_1st ROT Y SVD ERR
AND NOT   M0163A	// R_1st ROT Y STOP
AND NOT   M00733	// R_1st ROT Y NOT MV
AND NOT   M0163F	// R_1st ROT Y MOVE HOLD
OUT       M01630	// R_1st ROT Y READY
; L2
LOAD      M01630	// R_1st ROT Y READY
TON       T0513 0	// R_1st_13 Y READY
TON       T0713 20	// R_1st_13 Y READY 2s
; L4
LOAD NOT  M0163F	// R_1st ROT Y MOVE HOLD
AND NOT   M0313C	// R_1st_13 Y Pos HOME >
AND NOT   M01631	// R_1st_13 Y POWER ON
NOT
TON       T0613 3000	// R_1st_13 Y NOT MOVE
// output comment: Motor Not Move ¡ÆEAa
; L5
LOAD      M02130	// T)L_1st_05 Y HOME
LOAD NOT  M00730	// R_1st ROT Y NOT HOME
AND NOT   M00732	// R_1st ROT Y SVD ERR
NOT
AND       M00008	// LEFT RESET SW PLS
OR LOAD
AND       T0713	// R_1st_13 Y READY 2s
OR        M01631	// R_1st_13 Y POWER ON
AND NOT   M0313C	// R_1st_13 Y Pos HOME >
AND       D001240.2	// R_1st ROT Y SVD ON
AND NOT   M01633	// R_1st ROT Y HOME PLS
AND NOT   M00733	// R_1st ROT Y NOT MV
AND       T4204	// R_1st SS MANDREL BW
OUT       M01631	// R_1st_13 Y POWER ON
; L8
LOAD      M01631	// R_1st_13 Y POWER ON
AND       T0713	// R_1st_13 Y READY 2s
OR        M0313C	// R_1st_13 Y Pos HOME >
AND NOT   T0413	// R_1st ROT Y GOINIT->
AND       D001240.2	// R_1st ROT Y SVD ON
AND NOT   D002240.E	// R_1st ROT Y ¨¬n¡íoA¢´Ao
AND NOT   M01633	// R_1st ROT Y HOME PLS
AND NOT   M00732	// R_1st ROT Y SVD ERR
AND NOT   M00733	// R_1st ROT Y NOT MV
AND       M01232	// SYSTEM LEFT READY
AND       T4204	// R_1st SS MANDREL BW
OUT       M0313C	// R_1st_13 Y Pos HOME >
; L10
LOAD      M01633	// R_1st ROT Y HOME PLS
OR        M01632	// R_1st_13 Y HOME GOOD
AND NOT   M01631	// R_1st_13 Y POWER ON
AND NOT   M0313C	// R_1st_13 Y Pos HOME >
AND NOT   D002240.E	// R_1st ROT Y ¨¬n¡íoA¢´Ao
AND NOT   M00600	// EMERGENCY ALARM
OUT       M01632	// R_1st_13 Y HOME GOOD
; L12
LOAD      D001240.8	// R_1st ROT Y ¢¯©ªA¢®¢¯I¡¤a
OUTP      M01633	// R_1st ROT Y HOME PLS

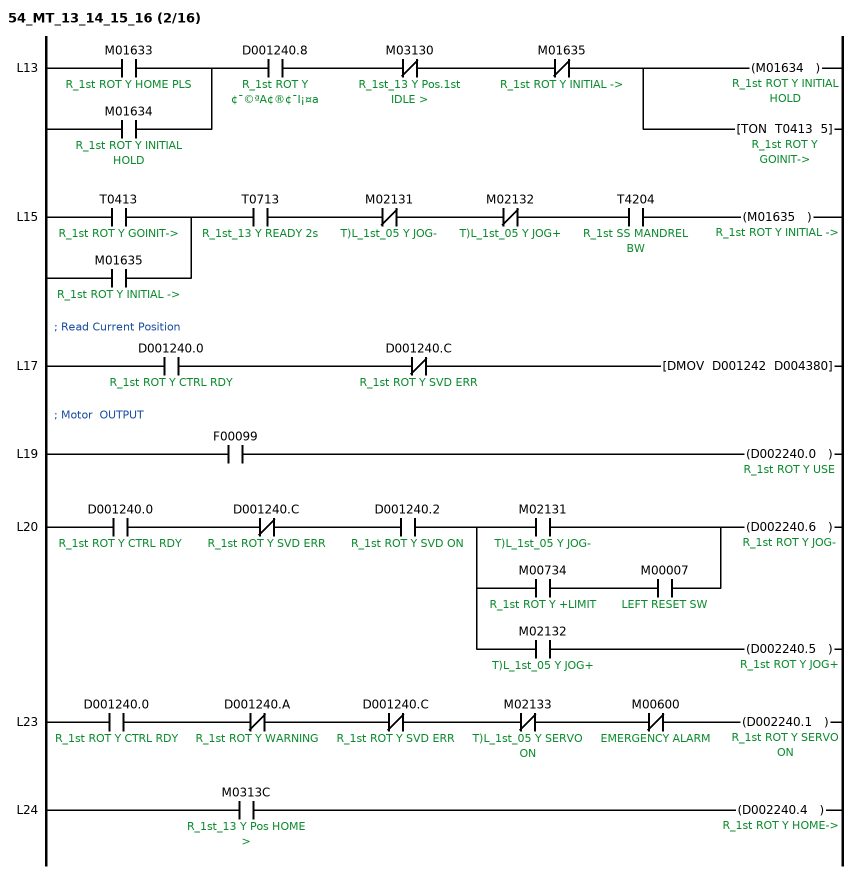
; L13
LOAD      M01633	// R_1st ROT Y HOME PLS
OR        M01634	// R_1st ROT Y INITIAL HOLD
AND       D001240.8	// R_1st ROT Y ¢¯©ªA¢®¢¯I¡¤a
AND NOT   M03130	// R_1st_13 Y Pos.1st IDLE >
AND NOT   M01635	// R_1st ROT Y INITIAL ->
OUT       M01634	// R_1st ROT Y INITIAL HOLD
TON       T0413 5	// R_1st ROT Y GOINIT->
; L15
LOAD      T0413	// R_1st ROT Y GOINIT->
OR        M01635	// R_1st ROT Y INITIAL ->
AND       T0713	// R_1st_13 Y READY 2s
AND NOT   M02131	// T)L_1st_05 Y JOG-
AND NOT   M02132	// T)L_1st_05 Y JOG+
AND       T4204	// R_1st SS MANDREL BW
OUT       M01635	// R_1st ROT Y INITIAL ->
; L17
LOAD      D001240.0	// R_1st ROT Y CTRL RDY
AND NOT   D001240.C	// R_1st ROT Y SVD ERR
DMOV      D001242 D004380
// output comment: Read Current Position
//  Motor  OUTPUT
; L19
LOAD      F00099
OUT       D002240.0	// R_1st ROT Y USE
; L20
LOAD      D001240.0	// R_1st ROT Y CTRL RDY
AND NOT   D001240.C	// R_1st ROT Y SVD ERR
AND       D001240.2	// R_1st ROT Y SVD ON
MPUSH
LOAD      M02131	// T)L_1st_05 Y JOG-
LOAD      M00734	// R_1st ROT Y +LIMIT
AND       M00007	// LEFT RESET SW
OR LOAD
AND LOAD
OUT       D002240.6	// R_1st ROT Y JOG-
MPOP
AND       M02132	// T)L_1st_05 Y JOG+
OUT       D002240.5	// R_1st ROT Y JOG+
; L23
LOAD      D001240.0	// R_1st ROT Y CTRL RDY
AND NOT   D001240.A	// R_1st ROT Y WARNING
AND NOT   D001240.C	// R_1st ROT Y SVD ERR
AND NOT   M02133	// T)L_1st_05 Y SERVO ON
AND NOT   M00600	// EMERGENCY ALARM
OUT       D002240.1	// R_1st ROT Y SERVO ON
; L24
LOAD      M0313C	// R_1st_13 Y Pos HOME >
OUT       D002240.4	// R_1st ROT Y HOME->

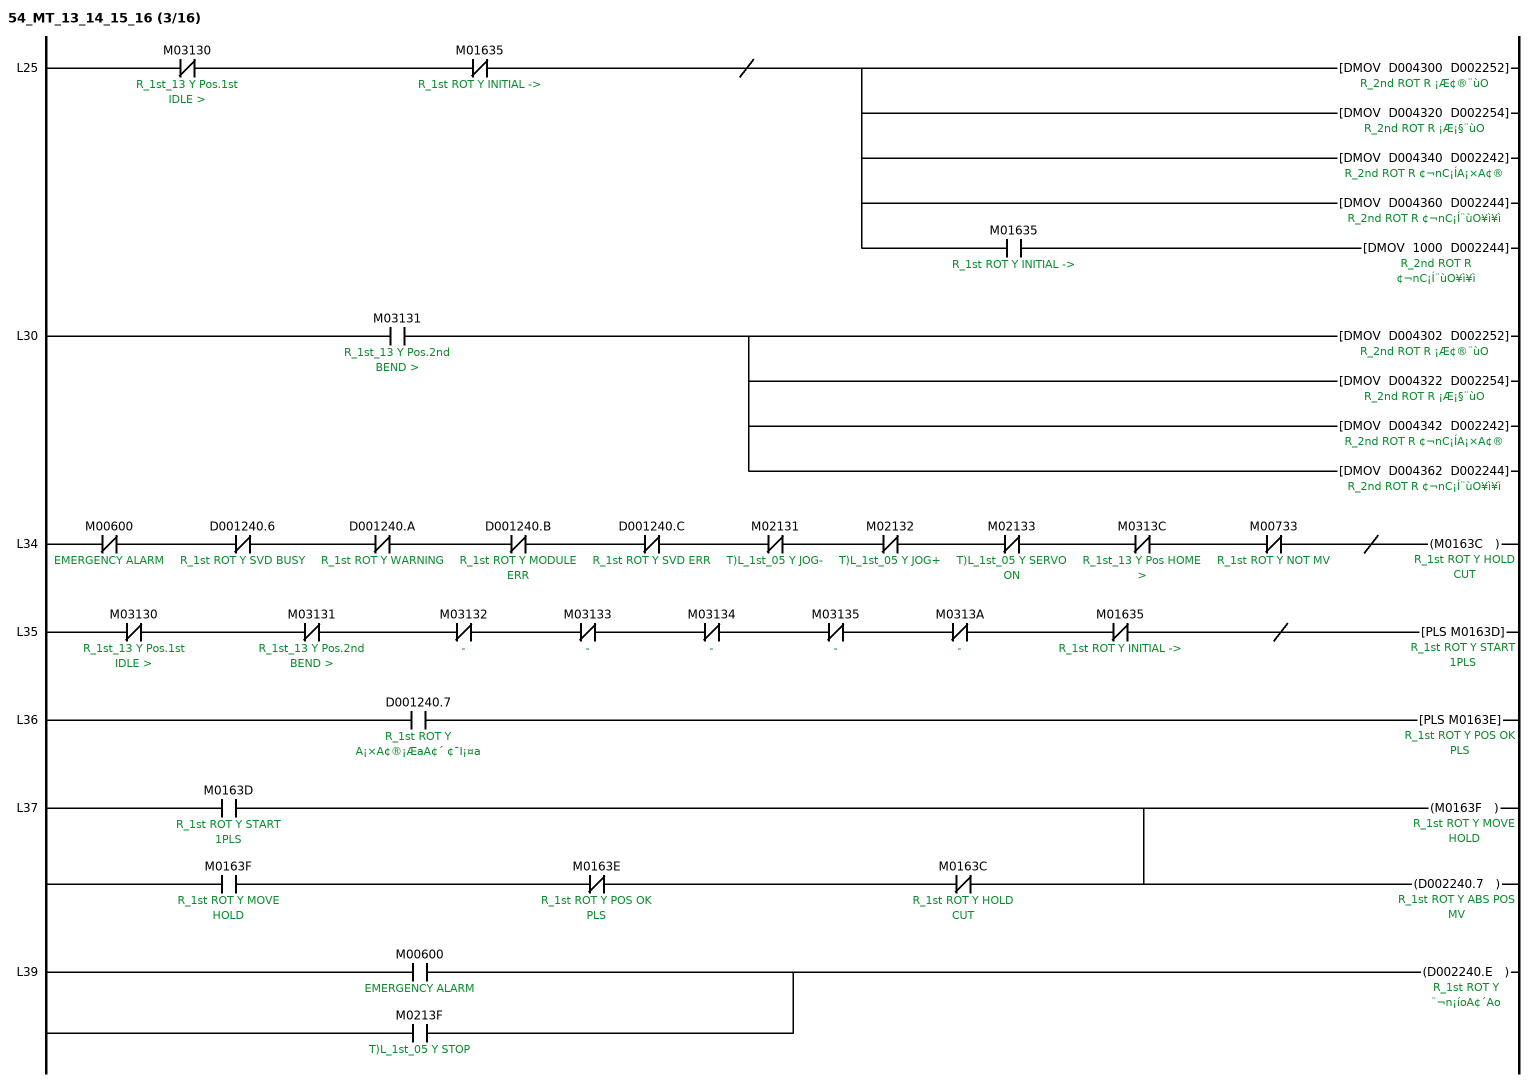
; L25
LOAD NOT  M03130	// R_1st_13 Y Pos.1st IDLE >
AND NOT   M01635	// R_1st ROT Y INITIAL ->
NOT
DMOV      D004300 D002252	// R_2nd ROT R ¡Æ¢®¨ùO
DMOV      D004320 D002254	// R_2nd ROT R ¡Æ¡§¨ùO
DMOV      D004340 D002242	// R_2nd ROT R ¢¬nC¡ÍA¡×A¢®
DMOV      D004360 D002244	// R_2nd ROT R ¢¬nC¡Í¨ùO¥ì¥ì
AND       M01635	// R_1st ROT Y INITIAL ->
DMOV      1000 D002244	// R_2nd ROT R ¢¬nC¡Í¨ùO¥ì¥ì
; L30
LOAD      M03131	// R_1st_13 Y Pos.2nd BEND >
DMOV      D004302 D002252	// R_2nd ROT R ¡Æ¢®¨ùO
DMOV      D004322 D002254	// R_2nd ROT R ¡Æ¡§¨ùO
DMOV      D004342 D002242	// R_2nd ROT R ¢¬nC¡ÍA¡×A¢®
DMOV      D004362 D002244	// R_2nd ROT R ¢¬nC¡Í¨ùO¥ì¥ì
; L34
LOAD NOT  M00600	// EMERGENCY ALARM
AND NOT   D001240.6	// R_1st ROT Y SVD BUSY
AND NOT   D001240.A	// R_1st ROT Y WARNING
AND NOT   D001240.B	// R_1st ROT Y MODULE ERR
AND NOT   D001240.C	// R_1st ROT Y SVD ERR
AND NOT   M02131	// T)L_1st_05 Y JOG-
AND NOT   M02132	// T)L_1st_05 Y JOG+
AND NOT   M02133	// T)L_1st_05 Y SERVO ON
AND NOT   M0313C	// R_1st_13 Y Pos HOME >
AND NOT   M00733	// R_1st ROT Y NOT MV
NOT
OUT       M0163C	// R_1st ROT Y HOLD CUT
; L35
LOAD NOT  M03130	// R_1st_13 Y Pos.1st IDLE >
AND NOT   M03131	// R_1st_13 Y Pos.2nd BEND >
AND NOT   M03132	// -
AND NOT   M03133	// -
AND NOT   M03134	// -
AND NOT   M03135	// -
AND NOT   M0313A	// -
AND NOT   M01635	// R_1st ROT Y INITIAL ->
NOT
OUTP      M0163D	// R_1st ROT Y START 1PLS
; L36
LOAD      D001240.7	// R_1st ROT Y A¡×A¢®¡ÆaA¢´ ¢¯I¡¤a
OUTP      M0163E	// R_1st ROT Y POS OK PLS
; L37
LOAD      M0163D	// R_1st ROT Y START 1PLS
LOAD      M0163F	// R_1st ROT Y MOVE HOLD
AND NOT   M0163E	// R_1st ROT Y POS OK PLS
AND NOT   M0163C	// R_1st ROT Y HOLD CUT
OR LOAD
OUT       M0163F	// R_1st ROT Y MOVE HOLD
OUT       D002240.7	// R_1st ROT Y ABS POS MV
; L39
LOAD      M00600	// EMERGENCY ALARM
OR        M0213F	// T)L_1st_05 Y STOP
OUT       D002240.E	// R_1st ROT Y ¨¬n¡íoA¢´Ao

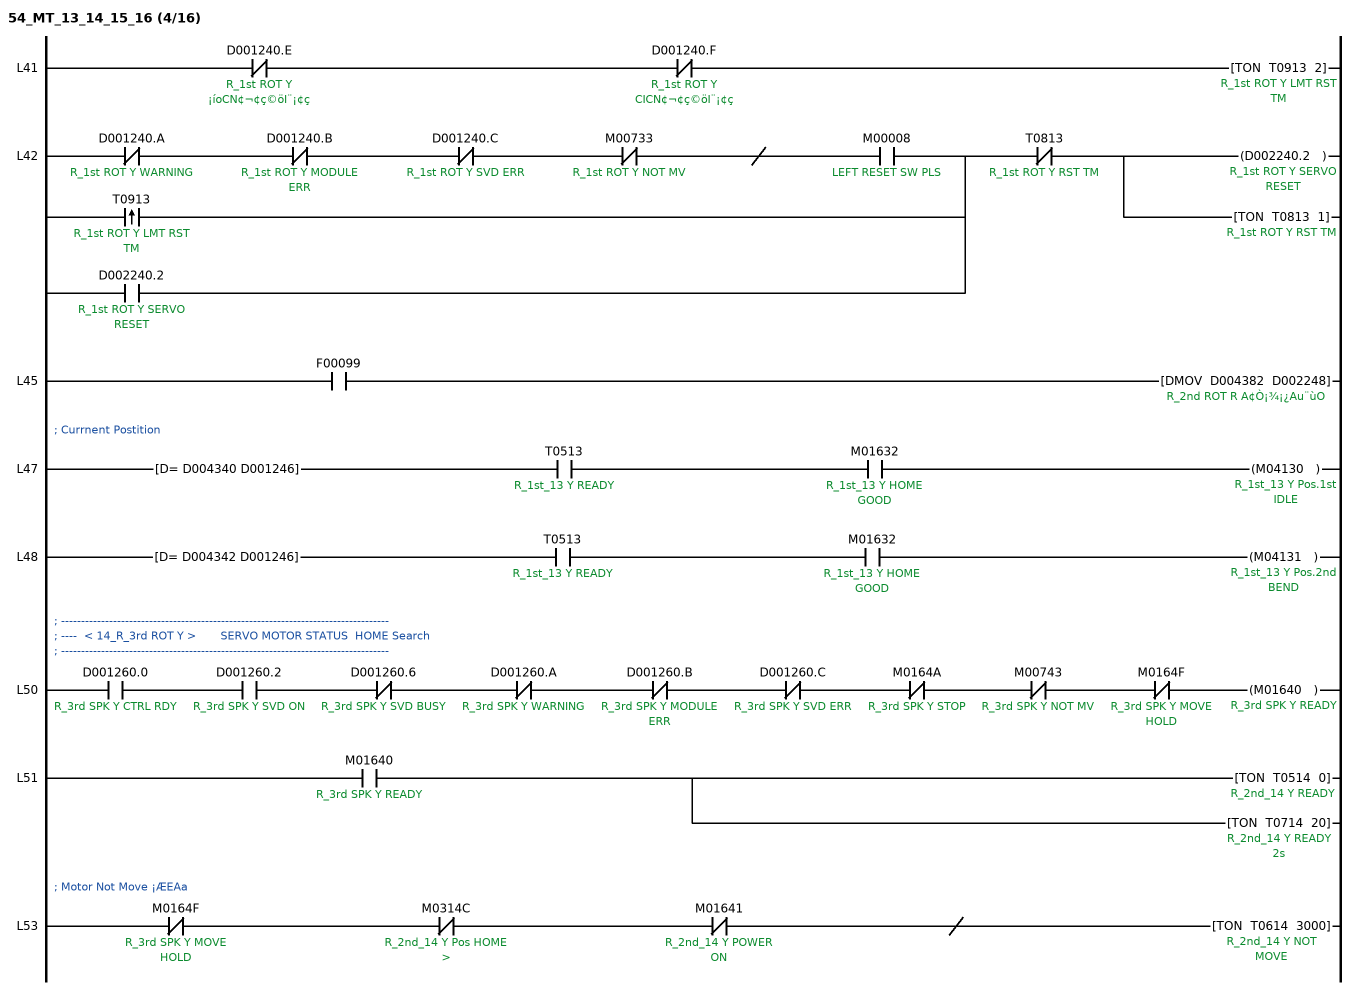
; L41
LOAD NOT  D001240.E	// R_1st ROT Y ¡íoCN¢¬¢ç©öI¨¡¢ç
AND NOT   D001240.F	// R_1st ROT Y CICN¢¬¢ç©öI¨¡¢ç
TON       T0913 2	// R_1st ROT Y LMT RST TM
; L42
LOAD NOT  D001240.A	// R_1st ROT Y WARNING
AND NOT   D001240.B	// R_1st ROT Y MODULE ERR
AND NOT   D001240.C	// R_1st ROT Y SVD ERR
AND NOT   M00733	// R_1st ROT Y NOT MV
NOT
AND       M00008	// LEFT RESET SW PLS
ORP       T0913	// R_1st ROT Y LMT RST TM
OR        D002240.2	// R_1st ROT Y SERVO RESET
AND NOT   T0813	// R_1st ROT Y RST TM
OUT       D002240.2	// R_1st ROT Y SERVO RESET
TON       T0813 1	// R_1st ROT Y RST TM
; L45
LOAD      F00099
DMOV      D004382 D002248	// R_2nd ROT R A¢Ò¡¾¡¿Au¨ùO
// Currnent Postition
; L47
LOADD=    D004340 D001246
AND       T0513	// R_1st_13 Y READY
AND       M01632	// R_1st_13 Y HOME GOOD
OUT       M04130	// R_1st_13 Y Pos.1st IDLE
; L48
LOADD=    D004342 D001246
AND       T0513	// R_1st_13 Y READY
AND       M01632	// R_1st_13 Y HOME GOOD
OUT       M04131	// R_1st_13 Y Pos.2nd BEND
// ----------------------------------------------------------------------------------
// 
// ----  < 14_R_3rd ROT Y >       SERVO MOTOR STATUS  HOME Search
// 
// ----------------------------------------------------------------------------------
; L50
LOAD      D001260.0	// R_3rd SPK Y CTRL RDY
AND       D001260.2	// R_3rd SPK Y SVD ON
AND NOT   D001260.6	// R_3rd SPK Y SVD BUSY
AND NOT   D001260.A	// R_3rd SPK Y WARNING
AND NOT   D001260.B	// R_3rd SPK Y MODULE ERR
AND NOT   D001260.C	// R_3rd SPK Y SVD ERR
AND NOT   M0164A	// R_3rd SPK Y STOP
AND NOT   M00743	// R_3rd SPK Y NOT MV
AND NOT   M0164F	// R_3rd SPK Y MOVE HOLD
OUT       M01640	// R_3rd SPK Y READY
; L51
LOAD      M01640	// R_3rd SPK Y READY
TON       T0514 0	// R_2nd_14 Y READY
TON       T0714 20	// R_2nd_14 Y READY 2s
; L53
LOAD NOT  M0164F	// R_3rd SPK Y MOVE HOLD
AND NOT   M0314C	// R_2nd_14 Y Pos HOME >
AND NOT   M01641	// R_2nd_14 Y POWER ON
NOT
TON       T0614 3000	// R_2nd_14 Y NOT MOVE
// output comment: Motor Not Move ¡ÆEAa

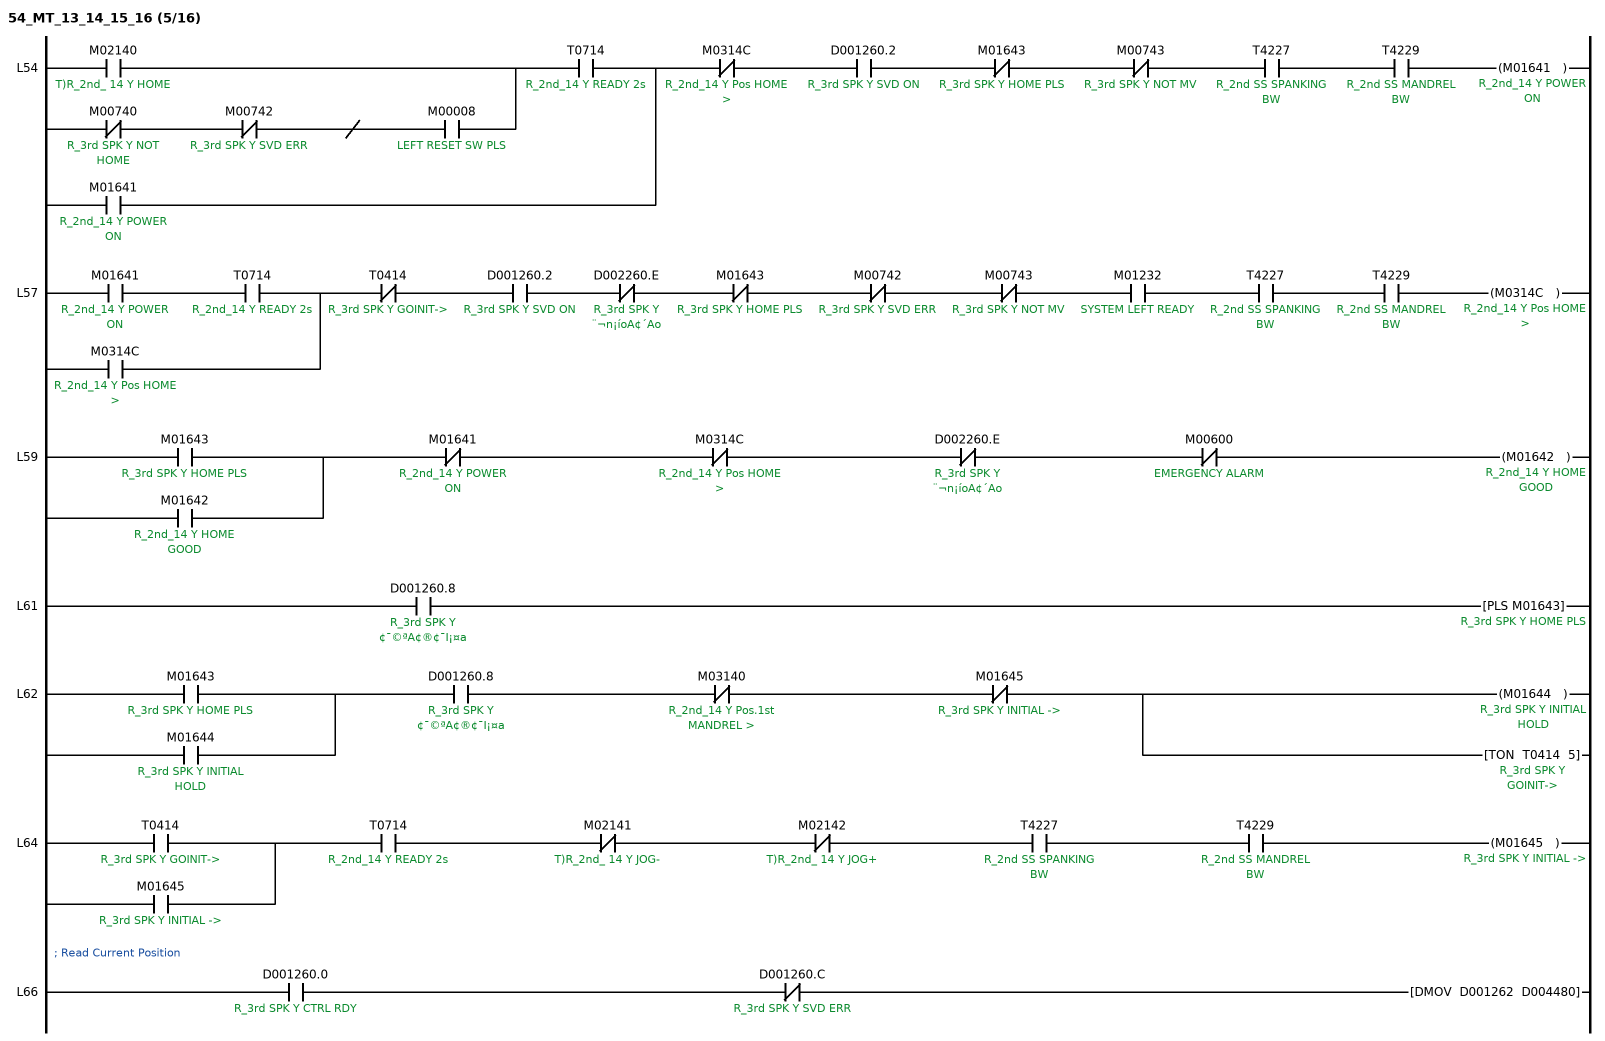
; L54
LOAD      M02140	// T)R_2nd_ 14 Y HOME
LOAD NOT  M00740	// R_3rd SPK Y NOT HOME
AND NOT   M00742	// R_3rd SPK Y SVD ERR
NOT
AND       M00008	// LEFT RESET SW PLS
OR LOAD
AND       T0714	// R_2nd_14 Y READY 2s
OR        M01641	// R_2nd_14 Y POWER ON
AND NOT   M0314C	// R_2nd_14 Y Pos HOME >
AND       D001260.2	// R_3rd SPK Y SVD ON
AND NOT   M01643	// R_3rd SPK Y HOME PLS
AND NOT   M00743	// R_3rd SPK Y NOT MV
AND       T4227	// R_2nd SS SPANKING BW
AND       T4229	// R_2nd SS MANDREL BW
OUT       M01641	// R_2nd_14 Y POWER ON
; L57
LOAD      M01641	// R_2nd_14 Y POWER ON
AND       T0714	// R_2nd_14 Y READY 2s
OR        M0314C	// R_2nd_14 Y Pos HOME >
AND NOT   T0414	// R_3rd SPK Y GOINIT->
AND       D001260.2	// R_3rd SPK Y SVD ON
AND NOT   D002260.E	// R_3rd SPK Y ¨¬n¡íoA¢´Ao
AND NOT   M01643	// R_3rd SPK Y HOME PLS
AND NOT   M00742	// R_3rd SPK Y SVD ERR
AND NOT   M00743	// R_3rd SPK Y NOT MV
AND       M01232	// SYSTEM LEFT READY
AND       T4227	// R_2nd SS SPANKING BW
AND       T4229	// R_2nd SS MANDREL BW
OUT       M0314C	// R_2nd_14 Y Pos HOME >
; L59
LOAD      M01643	// R_3rd SPK Y HOME PLS
OR        M01642	// R_2nd_14 Y HOME GOOD
AND NOT   M01641	// R_2nd_14 Y POWER ON
AND NOT   M0314C	// R_2nd_14 Y Pos HOME >
AND NOT   D002260.E	// R_3rd SPK Y ¨¬n¡íoA¢´Ao
AND NOT   M00600	// EMERGENCY ALARM
OUT       M01642	// R_2nd_14 Y HOME GOOD
; L61
LOAD      D001260.8	// R_3rd SPK Y ¢¯©ªA¢®¢¯I¡¤a
OUTP      M01643	// R_3rd SPK Y HOME PLS
; L62
LOAD      M01643	// R_3rd SPK Y HOME PLS
OR        M01644	// R_3rd SPK Y INITIAL HOLD
AND       D001260.8	// R_3rd SPK Y ¢¯©ªA¢®¢¯I¡¤a
AND NOT   M03140	// R_2nd_14 Y Pos.1st MANDREL >
AND NOT   M01645	// R_3rd SPK Y INITIAL ->
OUT       M01644	// R_3rd SPK Y INITIAL HOLD
TON       T0414 5	// R_3rd SPK Y GOINIT->
; L64
LOAD      T0414	// R_3rd SPK Y GOINIT->
OR        M01645	// R_3rd SPK Y INITIAL ->
AND       T0714	// R_2nd_14 Y READY 2s
AND NOT   M02141	// T)R_2nd_ 14 Y JOG-
AND NOT   M02142	// T)R_2nd_ 14 Y JOG+
AND       T4227	// R_2nd SS SPANKING BW
AND       T4229	// R_2nd SS MANDREL BW
OUT       M01645	// R_3rd SPK Y INITIAL ->
; L66
LOAD      D001260.0	// R_3rd SPK Y CTRL RDY
AND NOT   D001260.C	// R_3rd SPK Y SVD ERR
DMOV      D001262 D004480
// output comment: Read Current Position

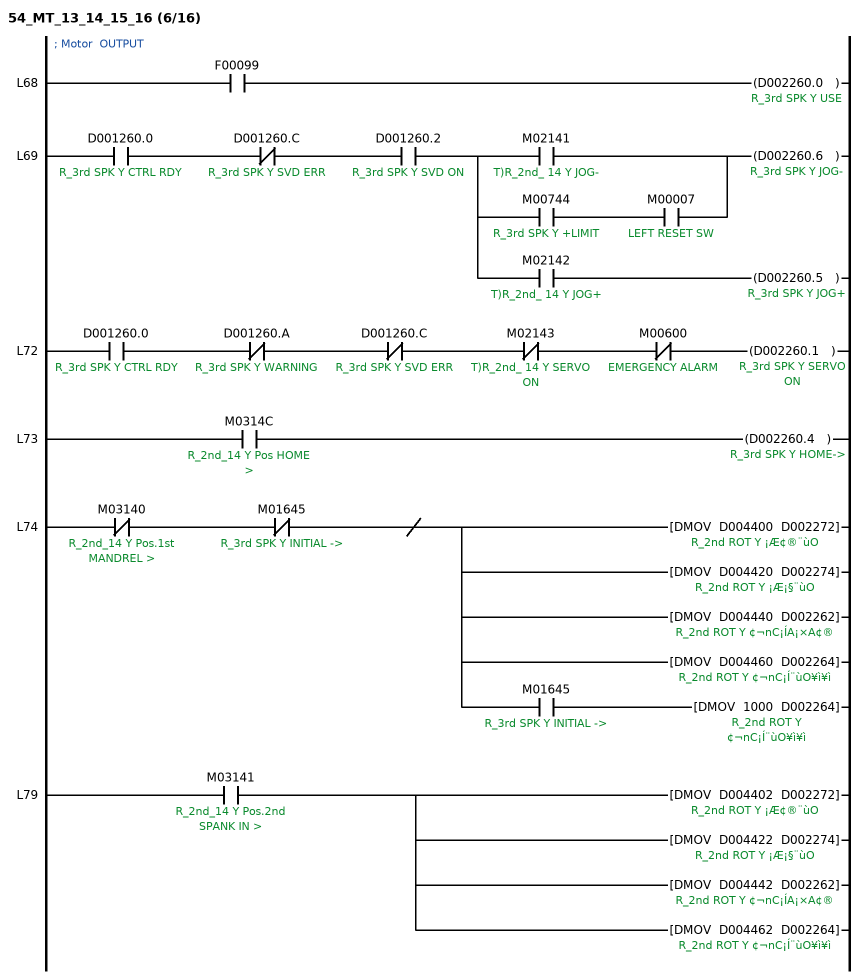
//  Motor  OUTPUT
; L68
LOAD      F00099
OUT       D002260.0	// R_3rd SPK Y USE
; L69
LOAD      D001260.0	// R_3rd SPK Y CTRL RDY
AND NOT   D001260.C	// R_3rd SPK Y SVD ERR
AND       D001260.2	// R_3rd SPK Y SVD ON
MPUSH
LOAD      M02141	// T)R_2nd_ 14 Y JOG-
LOAD      M00744	// R_3rd SPK Y +LIMIT
AND       M00007	// LEFT RESET SW
OR LOAD
AND LOAD
OUT       D002260.6	// R_3rd SPK Y JOG-
MPOP
AND       M02142	// T)R_2nd_ 14 Y JOG+
OUT       D002260.5	// R_3rd SPK Y JOG+
; L72
LOAD      D001260.0	// R_3rd SPK Y CTRL RDY
AND NOT   D001260.A	// R_3rd SPK Y WARNING
AND NOT   D001260.C	// R_3rd SPK Y SVD ERR
AND NOT   M02143	// T)R_2nd_ 14 Y SERVO ON
AND NOT   M00600	// EMERGENCY ALARM
OUT       D002260.1	// R_3rd SPK Y SERVO ON
; L73
LOAD      M0314C	// R_2nd_14 Y Pos HOME >
OUT       D002260.4	// R_3rd SPK Y HOME->
; L74
LOAD NOT  M03140	// R_2nd_14 Y Pos.1st MANDREL >
AND NOT   M01645	// R_3rd SPK Y INITIAL ->
NOT
DMOV      D004400 D002272	// R_2nd ROT Y ¡Æ¢®¨ùO
DMOV      D004420 D002274	// R_2nd ROT Y ¡Æ¡§¨ùO
DMOV      D004440 D002262	// R_2nd ROT Y ¢¬nC¡ÍA¡×A¢®
DMOV      D004460 D002264	// R_2nd ROT Y ¢¬nC¡Í¨ùO¥ì¥ì
AND       M01645	// R_3rd SPK Y INITIAL ->
DMOV      1000 D002264	// R_2nd ROT Y ¢¬nC¡Í¨ùO¥ì¥ì
; L79
LOAD      M03141	// R_2nd_14 Y Pos.2nd SPANK IN >
DMOV      D004402 D002272	// R_2nd ROT Y ¡Æ¢®¨ùO
DMOV      D004422 D002274	// R_2nd ROT Y ¡Æ¡§¨ùO
DMOV      D004442 D002262	// R_2nd ROT Y ¢¬nC¡ÍA¡×A¢®
DMOV      D004462 D002264	// R_2nd ROT Y ¢¬nC¡Í¨ùO¥ì¥ì

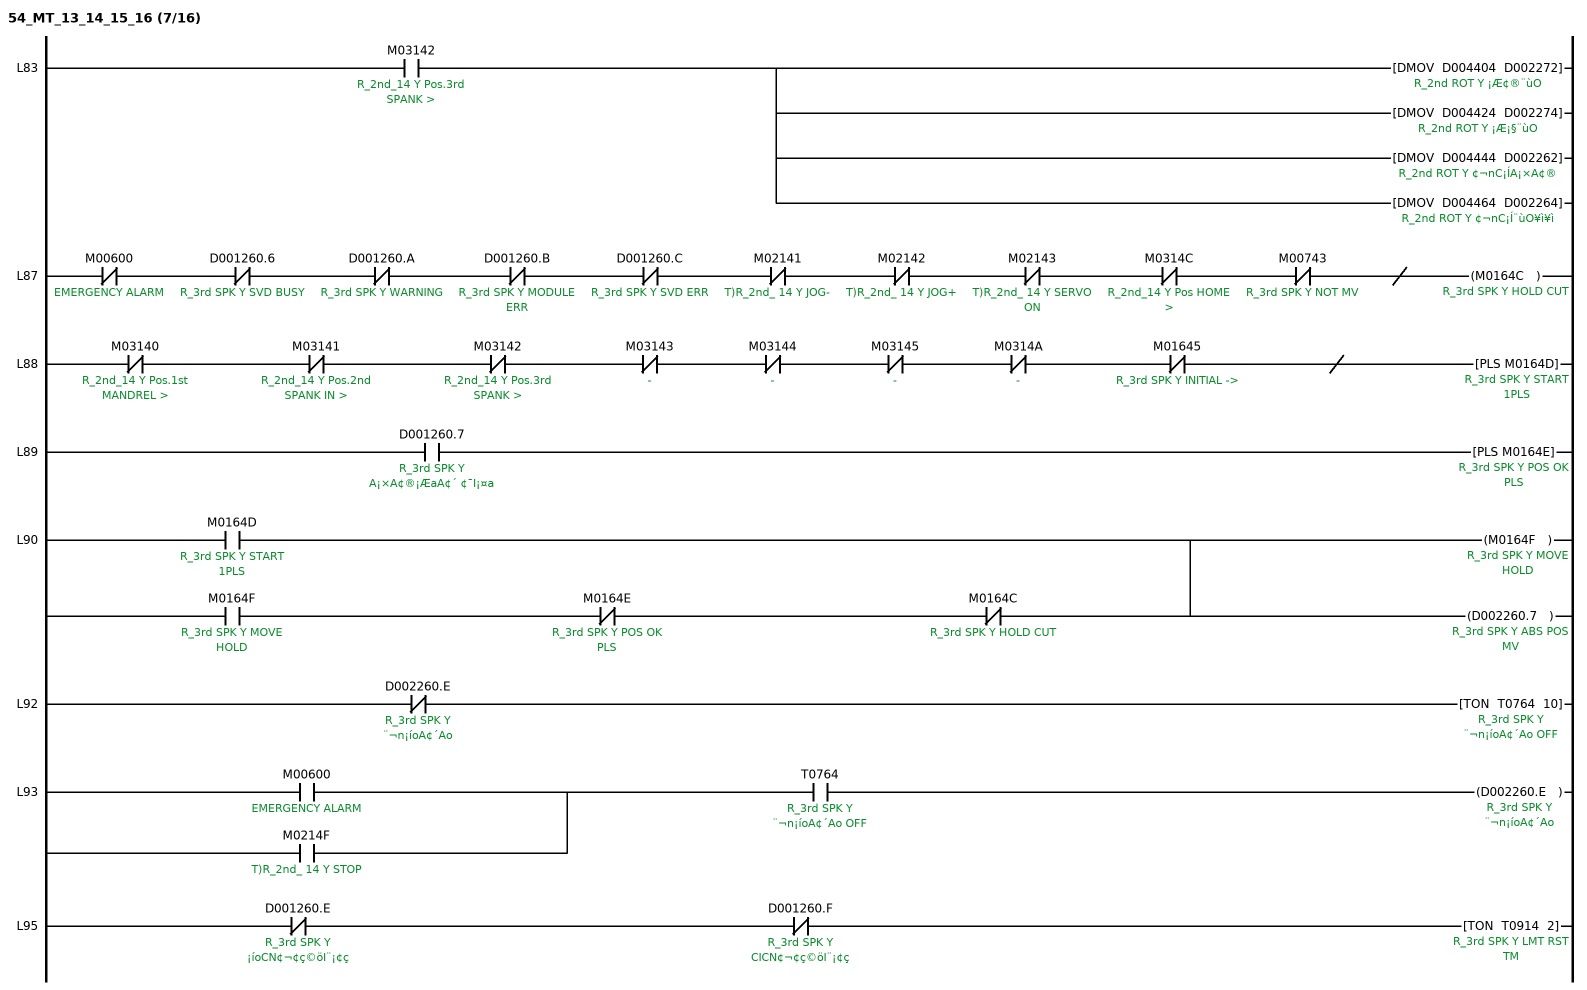
; L83
LOAD      M03142	// R_2nd_14 Y Pos.3rd SPANK >
DMOV      D004404 D002272	// R_2nd ROT Y ¡Æ¢®¨ùO
DMOV      D004424 D002274	// R_2nd ROT Y ¡Æ¡§¨ùO
DMOV      D004444 D002262	// R_2nd ROT Y ¢¬nC¡ÍA¡×A¢®
DMOV      D004464 D002264	// R_2nd ROT Y ¢¬nC¡Í¨ùO¥ì¥ì
; L87
LOAD NOT  M00600	// EMERGENCY ALARM
AND NOT   D001260.6	// R_3rd SPK Y SVD BUSY
AND NOT   D001260.A	// R_3rd SPK Y WARNING
AND NOT   D001260.B	// R_3rd SPK Y MODULE ERR
AND NOT   D001260.C	// R_3rd SPK Y SVD ERR
AND NOT   M02141	// T)R_2nd_ 14 Y JOG-
AND NOT   M02142	// T)R_2nd_ 14 Y JOG+
AND NOT   M02143	// T)R_2nd_ 14 Y SERVO ON
AND NOT   M0314C	// R_2nd_14 Y Pos HOME >
AND NOT   M00743	// R_3rd SPK Y NOT MV
NOT
OUT       M0164C	// R_3rd SPK Y HOLD CUT
; L88
LOAD NOT  M03140	// R_2nd_14 Y Pos.1st MANDREL >
AND NOT   M03141	// R_2nd_14 Y Pos.2nd SPANK IN >
AND NOT   M03142	// R_2nd_14 Y Pos.3rd SPANK >
AND NOT   M03143	// -
AND NOT   M03144	// -
AND NOT   M03145	// -
AND NOT   M0314A	// -
AND NOT   M01645	// R_3rd SPK Y INITIAL ->
NOT
OUTP      M0164D	// R_3rd SPK Y START 1PLS
; L89
LOAD      D001260.7	// R_3rd SPK Y A¡×A¢®¡ÆaA¢´ ¢¯I¡¤a
OUTP      M0164E	// R_3rd SPK Y POS OK PLS
; L90
LOAD      M0164D	// R_3rd SPK Y START 1PLS
LOAD      M0164F	// R_3rd SPK Y MOVE HOLD
AND NOT   M0164E	// R_3rd SPK Y POS OK PLS
AND NOT   M0164C	// R_3rd SPK Y HOLD CUT
OR LOAD
OUT       M0164F	// R_3rd SPK Y MOVE HOLD
OUT       D002260.7	// R_3rd SPK Y ABS POS MV
; L92
LOAD NOT  D002260.E	// R_3rd SPK Y ¨¬n¡íoA¢´Ao
TON       T0764 10	// R_3rd SPK Y ¨¬n¡íoA¢´Ao OFF
; L93
LOAD      M00600	// EMERGENCY ALARM
OR        M0214F	// T)R_2nd_ 14 Y STOP
AND       T0764	// R_3rd SPK Y ¨¬n¡íoA¢´Ao OFF
OUT       D002260.E	// R_3rd SPK Y ¨¬n¡íoA¢´Ao
; L95
LOAD NOT  D001260.E	// R_3rd SPK Y ¡íoCN¢¬¢ç©öI¨¡¢ç
AND NOT   D001260.F	// R_3rd SPK Y CICN¢¬¢ç©öI¨¡¢ç
TON       T0914 2	// R_3rd SPK Y LMT RST TM

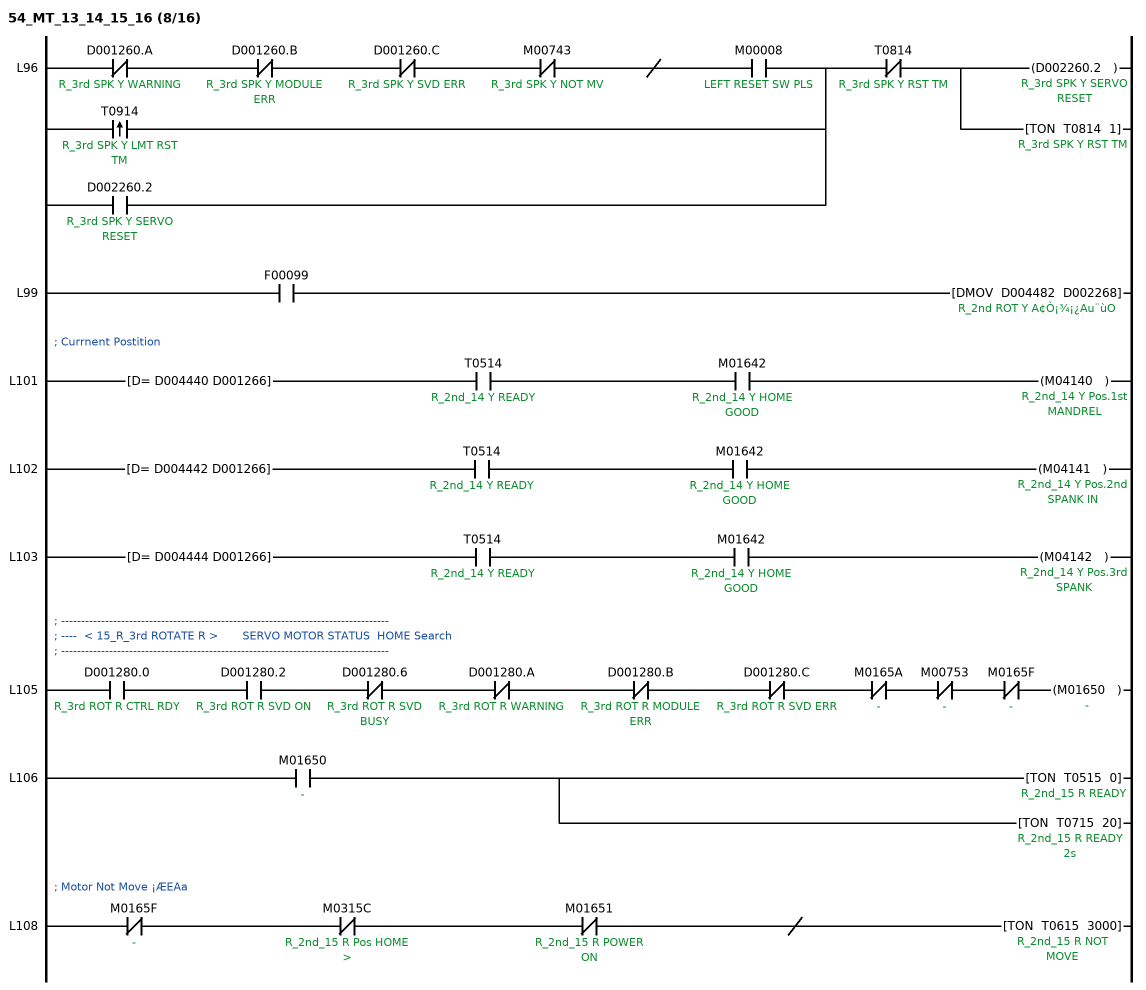
; L96
LOAD NOT  D001260.A	// R_3rd SPK Y WARNING
AND NOT   D001260.B	// R_3rd SPK Y MODULE ERR
AND NOT   D001260.C	// R_3rd SPK Y SVD ERR
AND NOT   M00743	// R_3rd SPK Y NOT MV
NOT
AND       M00008	// LEFT RESET SW PLS
ORP       T0914	// R_3rd SPK Y LMT RST TM
OR        D002260.2	// R_3rd SPK Y SERVO RESET
AND NOT   T0814	// R_3rd SPK Y RST TM
OUT       D002260.2	// R_3rd SPK Y SERVO RESET
TON       T0814 1	// R_3rd SPK Y RST TM
; L99
LOAD      F00099
DMOV      D004482 D002268	// R_2nd ROT Y A¢Ò¡¾¡¿Au¨ùO
// Currnent Postition
; L101
LOADD=    D004440 D001266
AND       T0514	// R_2nd_14 Y READY
AND       M01642	// R_2nd_14 Y HOME GOOD
OUT       M04140	// R_2nd_14 Y Pos.1st MANDREL
; L102
LOADD=    D004442 D001266
AND       T0514	// R_2nd_14 Y READY
AND       M01642	// R_2nd_14 Y HOME GOOD
OUT       M04141	// R_2nd_14 Y Pos.2nd SPANK IN
; L103
LOADD=    D004444 D001266
AND       T0514	// R_2nd_14 Y READY
AND       M01642	// R_2nd_14 Y HOME GOOD
OUT       M04142	// R_2nd_14 Y Pos.3rd SPANK
// ----------------------------------------------------------------------------------
// 
// ----  < 15_R_3rd ROTATE R >       SERVO MOTOR STATUS  HOME Search
// 
// ----------------------------------------------------------------------------------
; L105
LOAD      D001280.0	// R_3rd ROT R CTRL RDY
AND       D001280.2	// R_3rd ROT R SVD ON
AND NOT   D001280.6	// R_3rd ROT R SVD BUSY
AND NOT   D001280.A	// R_3rd ROT R WARNING
AND NOT   D001280.B	// R_3rd ROT R MODULE ERR
AND NOT   D001280.C	// R_3rd ROT R SVD ERR
AND NOT   M0165A	// -
AND NOT   M00753	// -
AND NOT   M0165F	// -
OUT       M01650	// -
; L106
LOAD      M01650	// -
TON       T0515 0	// R_2nd_15 R READY
TON       T0715 20	// R_2nd_15 R READY 2s
; L108
LOAD NOT  M0165F	// -
AND NOT   M0315C	// R_2nd_15 R Pos HOME >
AND NOT   M01651	// R_2nd_15 R POWER ON
NOT
TON       T0615 3000	// R_2nd_15 R NOT MOVE
// output comment: Motor Not Move ¡ÆEAa

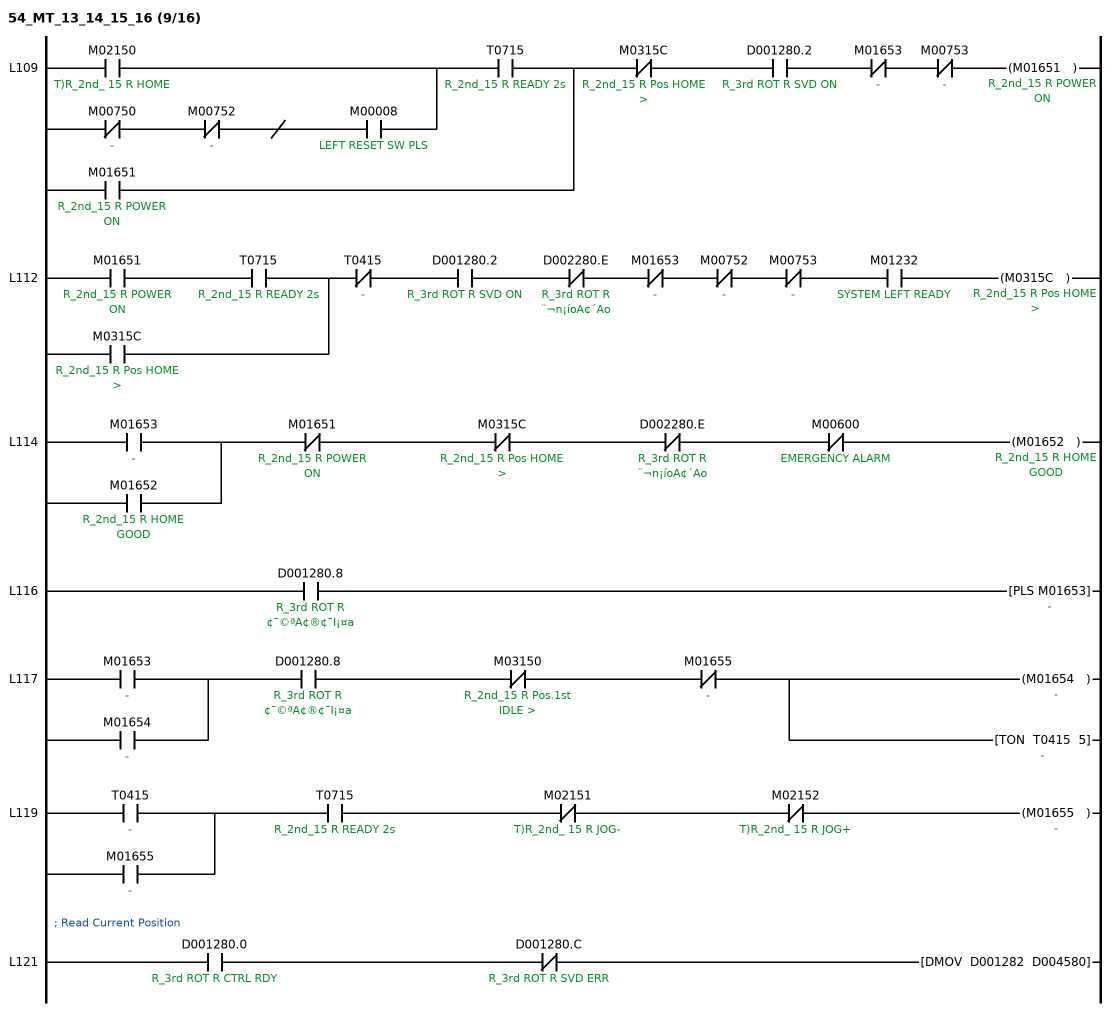
; L109
LOAD      M02150	// T)R_2nd_ 15 R HOME
LOAD NOT  M00750	// -
AND NOT   M00752	// -
NOT
AND       M00008	// LEFT RESET SW PLS
OR LOAD
AND       T0715	// R_2nd_15 R READY 2s
OR        M01651	// R_2nd_15 R POWER ON
AND NOT   M0315C	// R_2nd_15 R Pos HOME >
AND       D001280.2	// R_3rd ROT R SVD ON
AND NOT   M01653	// -
AND NOT   M00753	// -
OUT       M01651	// R_2nd_15 R POWER ON
; L112
LOAD      M01651	// R_2nd_15 R POWER ON
AND       T0715	// R_2nd_15 R READY 2s
OR        M0315C	// R_2nd_15 R Pos HOME >
AND NOT   T0415	// -
AND       D001280.2	// R_3rd ROT R SVD ON
AND NOT   D002280.E	// R_3rd ROT R ¨¬n¡íoA¢´Ao
AND NOT   M01653	// -
AND NOT   M00752	// -
AND NOT   M00753	// -
AND       M01232	// SYSTEM LEFT READY
OUT       M0315C	// R_2nd_15 R Pos HOME >
; L114
LOAD      M01653	// -
OR        M01652	// R_2nd_15 R HOME GOOD
AND NOT   M01651	// R_2nd_15 R POWER ON
AND NOT   M0315C	// R_2nd_15 R Pos HOME >
AND NOT   D002280.E	// R_3rd ROT R ¨¬n¡íoA¢´Ao
AND NOT   M00600	// EMERGENCY ALARM
OUT       M01652	// R_2nd_15 R HOME GOOD
; L116
LOAD      D001280.8	// R_3rd ROT R ¢¯©ªA¢®¢¯I¡¤a
OUTP      M01653	// -
; L117
LOAD      M01653	// -
OR        M01654	// -
AND       D001280.8	// R_3rd ROT R ¢¯©ªA¢®¢¯I¡¤a
AND NOT   M03150	// R_2nd_15 R Pos.1st IDLE >
AND NOT   M01655	// -
OUT       M01654	// -
TON       T0415 5	// -
; L119
LOAD      T0415	// -
OR        M01655	// -
AND       T0715	// R_2nd_15 R READY 2s
AND NOT   M02151	// T)R_2nd_ 15 R JOG-
AND NOT   M02152	// T)R_2nd_ 15 R JOG+
OUT       M01655	// -
; L121
LOAD      D001280.0	// R_3rd ROT R CTRL RDY
AND NOT   D001280.C	// R_3rd ROT R SVD ERR
DMOV      D001282 D004580
// output comment: Read Current Position

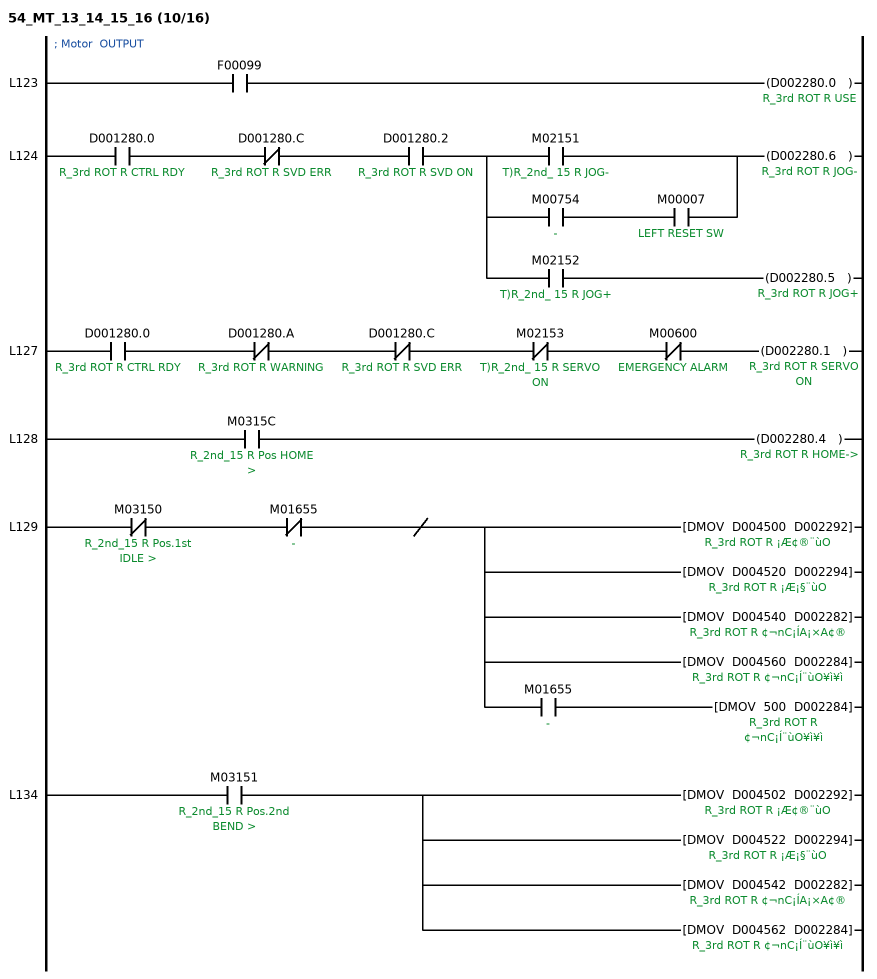
//  Motor  OUTPUT
; L123
LOAD      F00099
OUT       D002280.0	// R_3rd ROT R USE
; L124
LOAD      D001280.0	// R_3rd ROT R CTRL RDY
AND NOT   D001280.C	// R_3rd ROT R SVD ERR
AND       D001280.2	// R_3rd ROT R SVD ON
MPUSH
LOAD      M02151	// T)R_2nd_ 15 R JOG-
LOAD      M00754	// -
AND       M00007	// LEFT RESET SW
OR LOAD
AND LOAD
OUT       D002280.6	// R_3rd ROT R JOG-
MPOP
AND       M02152	// T)R_2nd_ 15 R JOG+
OUT       D002280.5	// R_3rd ROT R JOG+
; L127
LOAD      D001280.0	// R_3rd ROT R CTRL RDY
AND NOT   D001280.A	// R_3rd ROT R WARNING
AND NOT   D001280.C	// R_3rd ROT R SVD ERR
AND NOT   M02153	// T)R_2nd_ 15 R SERVO ON
AND NOT   M00600	// EMERGENCY ALARM
OUT       D002280.1	// R_3rd ROT R SERVO ON
; L128
LOAD      M0315C	// R_2nd_15 R Pos HOME >
OUT       D002280.4	// R_3rd ROT R HOME->
; L129
LOAD NOT  M03150	// R_2nd_15 R Pos.1st IDLE >
AND NOT   M01655	// -
NOT
DMOV      D004500 D002292	// R_3rd ROT R ¡Æ¢®¨ùO
DMOV      D004520 D002294	// R_3rd ROT R ¡Æ¡§¨ùO
DMOV      D004540 D002282	// R_3rd ROT R ¢¬nC¡ÍA¡×A¢®
DMOV      D004560 D002284	// R_3rd ROT R ¢¬nC¡Í¨ùO¥ì¥ì
AND       M01655	// -
DMOV      500 D002284	// R_3rd ROT R ¢¬nC¡Í¨ùO¥ì¥ì
; L134
LOAD      M03151	// R_2nd_15 R Pos.2nd BEND >
DMOV      D004502 D002292	// R_3rd ROT R ¡Æ¢®¨ùO
DMOV      D004522 D002294	// R_3rd ROT R ¡Æ¡§¨ùO
DMOV      D004542 D002282	// R_3rd ROT R ¢¬nC¡ÍA¡×A¢®
DMOV      D004562 D002284	// R_3rd ROT R ¢¬nC¡Í¨ùO¥ì¥ì

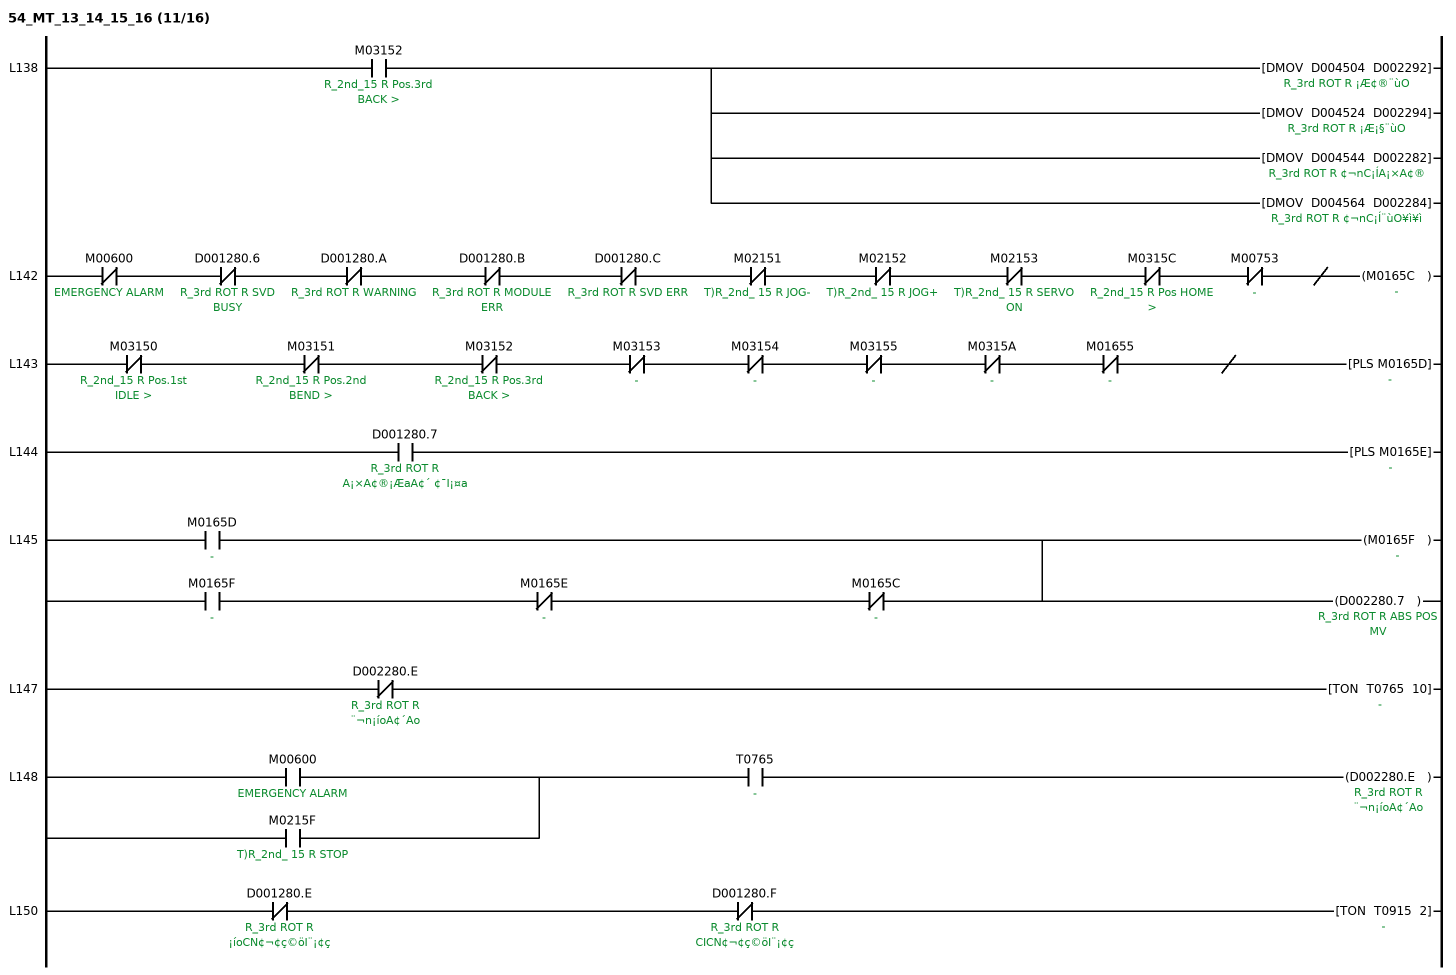
; L138
LOAD      M03152	// R_2nd_15 R Pos.3rd BACK >
DMOV      D004504 D002292	// R_3rd ROT R ¡Æ¢®¨ùO
DMOV      D004524 D002294	// R_3rd ROT R ¡Æ¡§¨ùO
DMOV      D004544 D002282	// R_3rd ROT R ¢¬nC¡ÍA¡×A¢®
DMOV      D004564 D002284	// R_3rd ROT R ¢¬nC¡Í¨ùO¥ì¥ì
; L142
LOAD NOT  M00600	// EMERGENCY ALARM
AND NOT   D001280.6	// R_3rd ROT R SVD BUSY
AND NOT   D001280.A	// R_3rd ROT R WARNING
AND NOT   D001280.B	// R_3rd ROT R MODULE ERR
AND NOT   D001280.C	// R_3rd ROT R SVD ERR
AND NOT   M02151	// T)R_2nd_ 15 R JOG-
AND NOT   M02152	// T)R_2nd_ 15 R JOG+
AND NOT   M02153	// T)R_2nd_ 15 R SERVO ON
AND NOT   M0315C	// R_2nd_15 R Pos HOME >
AND NOT   M00753	// -
NOT
OUT       M0165C	// -
; L143
LOAD NOT  M03150	// R_2nd_15 R Pos.1st IDLE >
AND NOT   M03151	// R_2nd_15 R Pos.2nd BEND >
AND NOT   M03152	// R_2nd_15 R Pos.3rd BACK >
AND NOT   M03153	// -
AND NOT   M03154	// -
AND NOT   M03155	// -
AND NOT   M0315A	// -
AND NOT   M01655	// -
NOT
OUTP      M0165D	// -
; L144
LOAD      D001280.7	// R_3rd ROT R A¡×A¢®¡ÆaA¢´ ¢¯I¡¤a
OUTP      M0165E	// -
; L145
LOAD      M0165D	// -
LOAD      M0165F	// -
AND NOT   M0165E	// -
AND NOT   M0165C	// -
OR LOAD
OUT       M0165F	// -
OUT       D002280.7	// R_3rd ROT R ABS POS MV
; L147
LOAD NOT  D002280.E	// R_3rd ROT R ¨¬n¡íoA¢´Ao
TON       T0765 10	// -
; L148
LOAD      M00600	// EMERGENCY ALARM
OR        M0215F	// T)R_2nd_ 15 R STOP
AND       T0765	// -
OUT       D002280.E	// R_3rd ROT R ¨¬n¡íoA¢´Ao
; L150
LOAD NOT  D001280.E	// R_3rd ROT R ¡íoCN¢¬¢ç©öI¨¡¢ç
AND NOT   D001280.F	// R_3rd ROT R CICN¢¬¢ç©öI¨¡¢ç
TON       T0915 2	// -

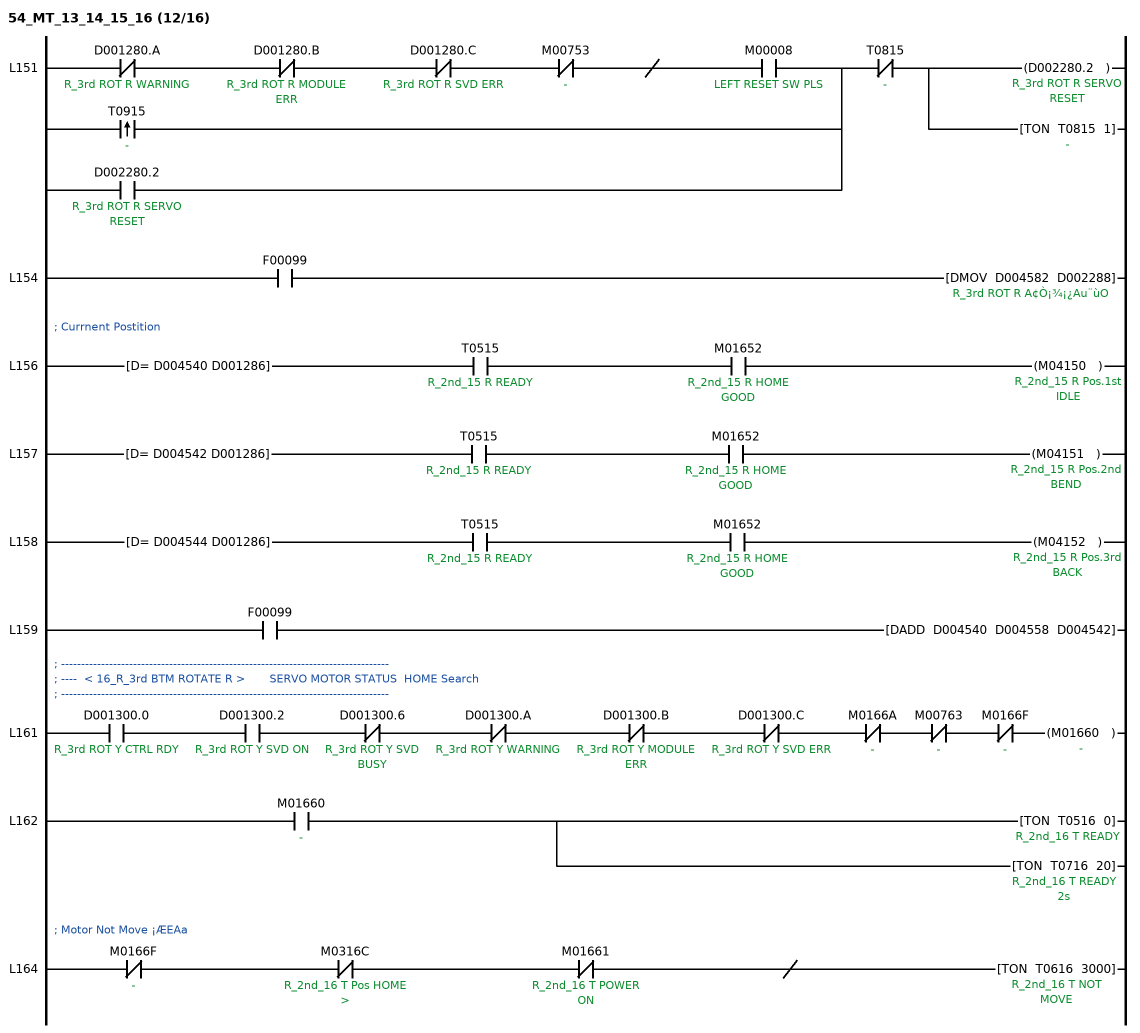
; L151
LOAD NOT  D001280.A	// R_3rd ROT R WARNING
AND NOT   D001280.B	// R_3rd ROT R MODULE ERR
AND NOT   D001280.C	// R_3rd ROT R SVD ERR
AND NOT   M00753	// -
NOT
AND       M00008	// LEFT RESET SW PLS
ORP       T0915	// -
OR        D002280.2	// R_3rd ROT R SERVO RESET
AND NOT   T0815	// -
OUT       D002280.2	// R_3rd ROT R SERVO RESET
TON       T0815 1	// -
; L154
LOAD      F00099
DMOV      D004582 D002288	// R_3rd ROT R A¢Ò¡¾¡¿Au¨ùO
// Currnent Postition
; L156
LOADD=    D004540 D001286
AND       T0515	// R_2nd_15 R READY
AND       M01652	// R_2nd_15 R HOME GOOD
OUT       M04150	// R_2nd_15 R Pos.1st IDLE
; L157
LOADD=    D004542 D001286
AND       T0515	// R_2nd_15 R READY
AND       M01652	// R_2nd_15 R HOME GOOD
OUT       M04151	// R_2nd_15 R Pos.2nd BEND
; L158
LOADD=    D004544 D001286
AND       T0515	// R_2nd_15 R READY
AND       M01652	// R_2nd_15 R HOME GOOD
OUT       M04152	// R_2nd_15 R Pos.3rd BACK
; L159
LOAD      F00099
DADD      D004540 D004558 D004542
// ----------------------------------------------------------------------------------
// 
// ----  < 16_R_3rd BTM ROTATE R >       SERVO MOTOR STATUS  HOME Search
// 
// ----------------------------------------------------------------------------------
; L161
LOAD      D001300.0	// R_3rd ROT Y CTRL RDY
AND       D001300.2	// R_3rd ROT Y SVD ON
AND NOT   D001300.6	// R_3rd ROT Y SVD BUSY
AND NOT   D001300.A	// R_3rd ROT Y WARNING
AND NOT   D001300.B	// R_3rd ROT Y MODULE ERR
AND NOT   D001300.C	// R_3rd ROT Y SVD ERR
AND NOT   M0166A	// -
AND NOT   M00763	// -
AND NOT   M0166F	// -
OUT       M01660	// -
; L162
LOAD      M01660	// -
TON       T0516 0	// R_2nd_16 T READY
TON       T0716 20	// R_2nd_16 T READY 2s
; L164
LOAD NOT  M0166F	// -
AND NOT   M0316C	// R_2nd_16 T Pos HOME >
AND NOT   M01661	// R_2nd_16 T POWER ON
NOT
TON       T0616 3000	// R_2nd_16 T NOT MOVE
// output comment: Motor Not Move ¡ÆEAa

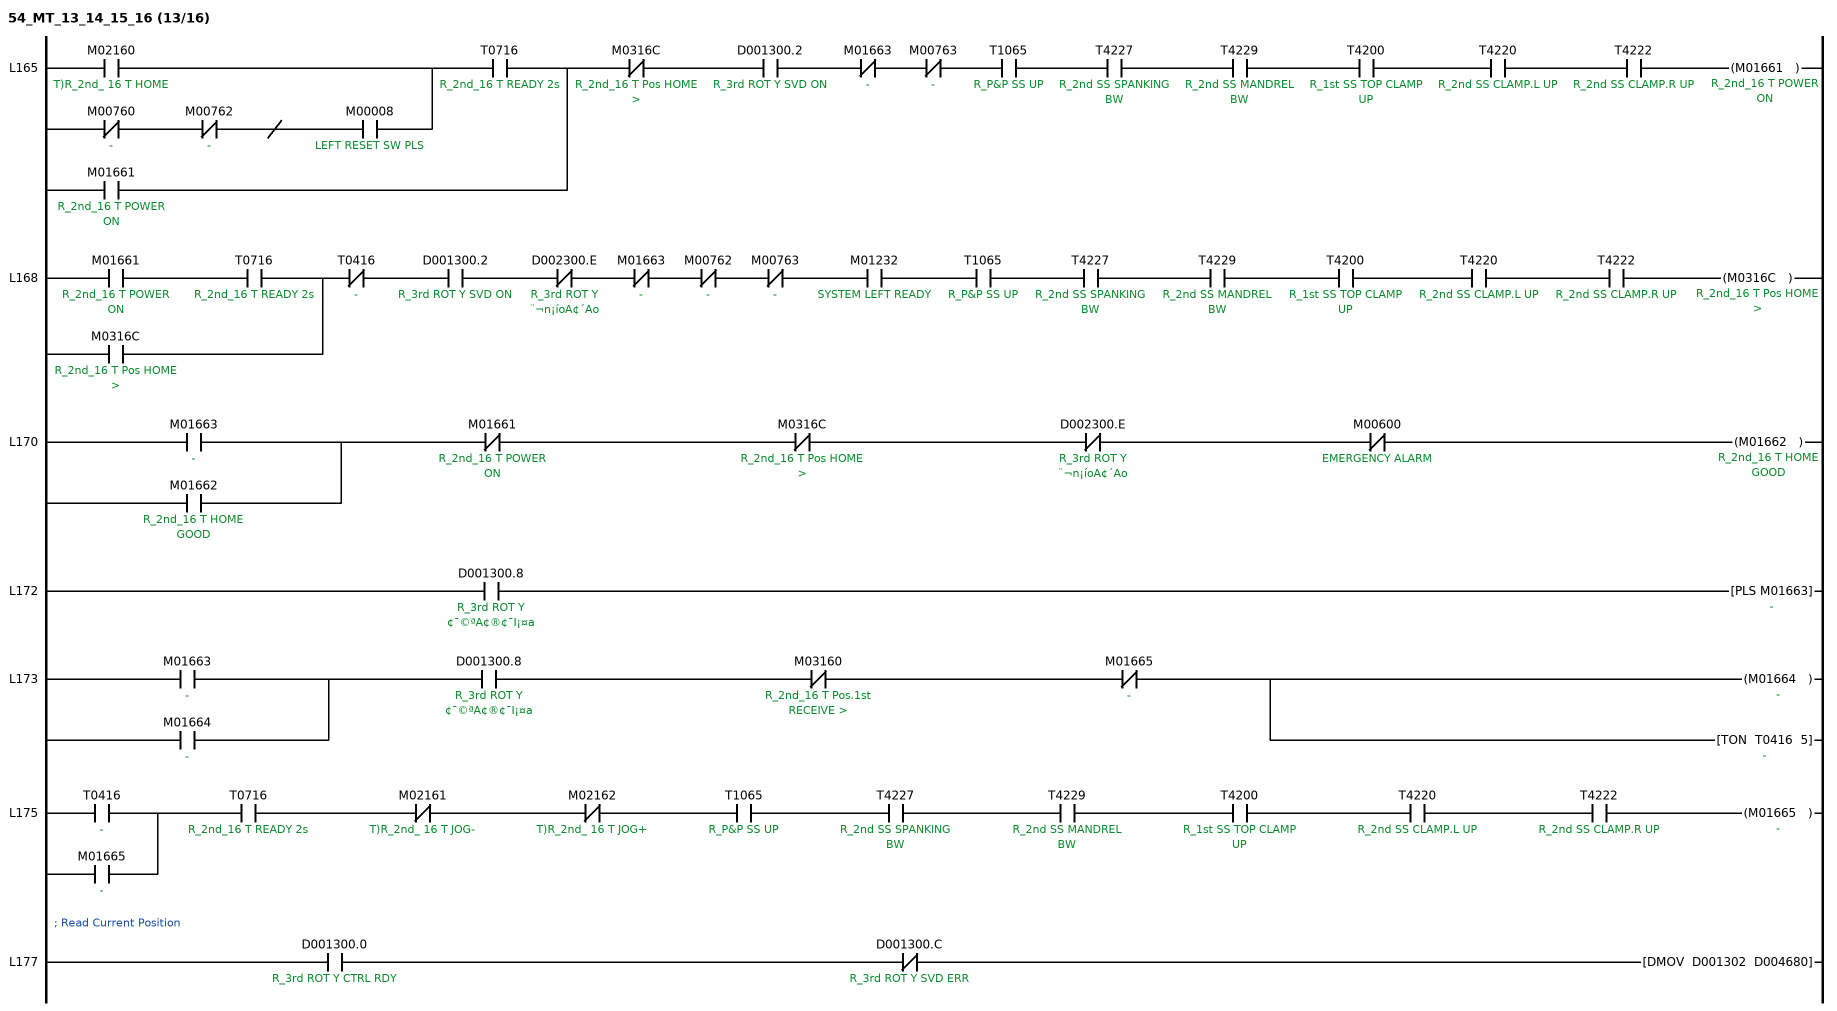
; L165
LOAD      M02160	// T)R_2nd_ 16 T HOME
LOAD NOT  M00760	// -
AND NOT   M00762	// -
NOT
AND       M00008	// LEFT RESET SW PLS
OR LOAD
AND       T0716	// R_2nd_16 T READY 2s
OR        M01661	// R_2nd_16 T POWER ON
AND NOT   M0316C	// R_2nd_16 T Pos HOME >
AND       D001300.2	// R_3rd ROT Y SVD ON
AND NOT   M01663	// -
AND NOT   M00763	// -
AND       T1065	// R_P&P SS UP
AND       T4227	// R_2nd SS SPANKING BW
AND       T4229	// R_2nd SS MANDREL BW
AND       T4200	// R_1st SS TOP CLAMP UP
AND       T4220	// R_2nd SS CLAMP.L UP
AND       T4222	// R_2nd SS CLAMP.R UP
OUT       M01661	// R_2nd_16 T POWER ON
; L168
LOAD      M01661	// R_2nd_16 T POWER ON
AND       T0716	// R_2nd_16 T READY 2s
OR        M0316C	// R_2nd_16 T Pos HOME >
AND NOT   T0416	// -
AND       D001300.2	// R_3rd ROT Y SVD ON
AND NOT   D002300.E	// R_3rd ROT Y ¨¬n¡íoA¢´Ao
AND NOT   M01663	// -
AND NOT   M00762	// -
AND NOT   M00763	// -
AND       M01232	// SYSTEM LEFT READY
AND       T1065	// R_P&P SS UP
AND       T4227	// R_2nd SS SPANKING BW
AND       T4229	// R_2nd SS MANDREL BW
AND       T4200	// R_1st SS TOP CLAMP UP
AND       T4220	// R_2nd SS CLAMP.L UP
AND       T4222	// R_2nd SS CLAMP.R UP
OUT       M0316C	// R_2nd_16 T Pos HOME >
; L170
LOAD      M01663	// -
OR        M01662	// R_2nd_16 T HOME GOOD
AND NOT   M01661	// R_2nd_16 T POWER ON
AND NOT   M0316C	// R_2nd_16 T Pos HOME >
AND NOT   D002300.E	// R_3rd ROT Y ¨¬n¡íoA¢´Ao
AND NOT   M00600	// EMERGENCY ALARM
OUT       M01662	// R_2nd_16 T HOME GOOD
; L172
LOAD      D001300.8	// R_3rd ROT Y ¢¯©ªA¢®¢¯I¡¤a
OUTP      M01663	// -
; L173
LOAD      M01663	// -
OR        M01664	// -
AND       D001300.8	// R_3rd ROT Y ¢¯©ªA¢®¢¯I¡¤a
AND NOT   M03160	// R_2nd_16 T Pos.1st RECEIVE >
AND NOT   M01665	// -
OUT       M01664	// -
TON       T0416 5	// -
; L175
LOAD      T0416	// -
OR        M01665	// -
AND       T0716	// R_2nd_16 T READY 2s
AND NOT   M02161	// T)R_2nd_ 16 T JOG-
AND NOT   M02162	// T)R_2nd_ 16 T JOG+
AND       T1065	// R_P&P SS UP
AND       T4227	// R_2nd SS SPANKING BW
AND       T4229	// R_2nd SS MANDREL BW
AND       T4200	// R_1st SS TOP CLAMP UP
AND       T4220	// R_2nd SS CLAMP.L UP
AND       T4222	// R_2nd SS CLAMP.R UP
OUT       M01665	// -
; L177
LOAD      D001300.0	// R_3rd ROT Y CTRL RDY
AND NOT   D001300.C	// R_3rd ROT Y SVD ERR
DMOV      D001302 D004680
// output comment: Read Current Position

